// TIA Portal V18 export
FUNCTION "ChangeOverProcess" : Void   // FC1000, LAD
{ S7_Optimized_Access := 'TRUE' }
// stored: AutoNumber false, SetENOAutomatically false
   VAR_TEMP
      tBool : Bool;
   END_VAR
   VAR_TEMP   // added for the SCL form of the ladder/FBD networks
      _w1 : Bool;
      _w2 : Bool;
      _w3 : Bool;
      _w4 : Bool;
      _w5 : Bool;
      _w6 : Bool;
      _w7 : Bool;
      _w8 : Bool;
   END_VAR
BEGIN

REGION Network 1: HMI ChangeOver Confirm
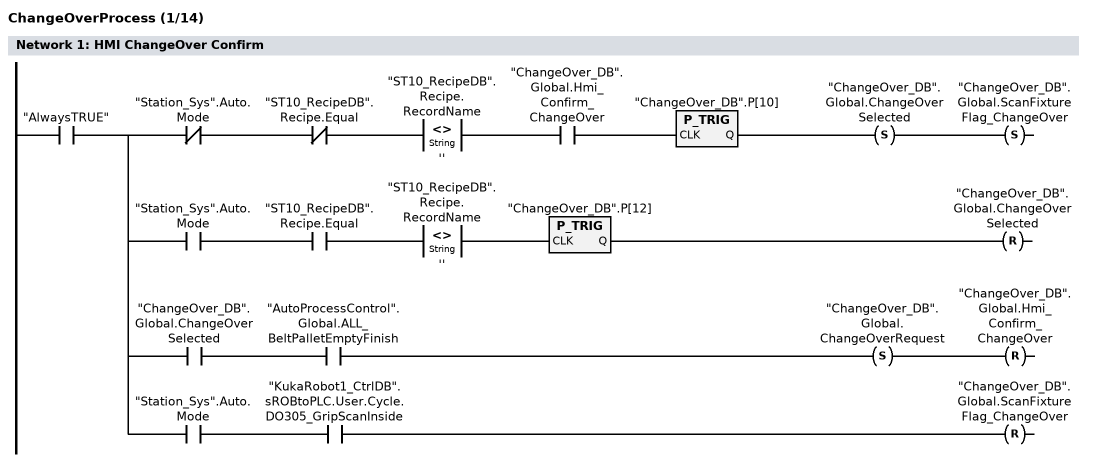
   RUNG wire#powerrail
      Contact( "AlwaysTRUE" )
      wire#w1
      I_Contact( "Station_Sys".Auto.Mode )
      I_Contact( "ST10_RecipeDB".Recipe.Equal )
      { S7_Templates := "SrcType := String" } NE_Contact(in1 := "ST10_RecipeDB".Recipe.RecordName, in2 := '')
      Contact( "ChangeOver_DB".Global.Hmi_Confirm_ChangeOver )
      P_Trig( "ChangeOver_DB".P[10] )
      S_Coil( "ChangeOver_DB".Global.ChangeOverSelected )
      S_Coil( "ChangeOver_DB".Global.ScanFixtureFlag_ChangeOver )
   END_RUNG
   RUNG wire#w1
      Contact( "Station_Sys".Auto.Mode )
      Contact( "ST10_RecipeDB".Recipe.Equal )
      { S7_Templates := "SrcType := String" } NE_Contact(in1 := "ST10_RecipeDB".Recipe.RecordName, in2 := '')
      P_Trig( "ChangeOver_DB".P[12] )
      R_Coil( "ChangeOver_DB".Global.ChangeOverSelected )
   END_RUNG
   RUNG wire#w1
      Contact( "ChangeOver_DB".Global.ChangeOverSelected )
      Contact( "AutoProcessControl".Global.ALL_BeltPalletEmptyFinish )
      S_Coil( "ChangeOver_DB".Global.ChangeOverRequest )
      R_Coil( "ChangeOver_DB".Global.Hmi_Confirm_ChangeOver )
   END_RUNG
   RUNG wire#w1
      Contact( "Station_Sys".Auto.Mode )
      Contact( "KukaRobot1_CtrlDB".sROBtoPLC.User.Cycle.DO305_GripScanInside )
      R_Coil( "ChangeOver_DB".Global.ScanFixtureFlag_ChangeOver )
   END_RUNG
   // the same network as SCL:
   #_w1 := "AlwaysTRUE" AND NOT "Station_Sys".Auto.Mode AND NOT "ST10_RecipeDB".Recipe.Equal AND ("ST10_RecipeDB".Recipe.RecordName <> '') AND "ChangeOver_DB".Global.Hmi_Confirm_ChangeOver;
   #_w2 := #_w1 AND NOT "ChangeOver_DB".P[10];   // rising edge
   "ChangeOver_DB".P[10] := #_w1;
   IF #_w2 THEN
       "ChangeOver_DB".Global.ChangeOverSelected := TRUE;
       "ChangeOver_DB".Global.ScanFixtureFlag_ChangeOver := TRUE;
   END_IF;
   #_w3 := "AlwaysTRUE" AND "Station_Sys".Auto.Mode AND "ST10_RecipeDB".Recipe.Equal AND ("ST10_RecipeDB".Recipe.RecordName <> '');
   #_w4 := #_w3 AND NOT "ChangeOver_DB".P[12];   // rising edge
   "ChangeOver_DB".P[12] := #_w3;
   IF #_w4 THEN "ChangeOver_DB".Global.ChangeOverSelected := FALSE; END_IF;
   IF "AlwaysTRUE" AND "ChangeOver_DB".Global.ChangeOverSelected AND "AutoProcessControl".Global.ALL_BeltPalletEmptyFinish THEN
       "ChangeOver_DB".Global.ChangeOverRequest := TRUE;
       "ChangeOver_DB".Global.Hmi_Confirm_ChangeOver := FALSE;
   END_IF;
   IF "AlwaysTRUE" AND "Station_Sys".Auto.Mode AND "KukaRobot1_CtrlDB".sROBtoPLC.User.Cycle.DO305_GripScanInside THEN
       "ChangeOver_DB".Global.ScanFixtureFlag_ChangeOver := FALSE;
   END_IF;
END_REGION

REGION Network 2: ChangeOverFinish Reset
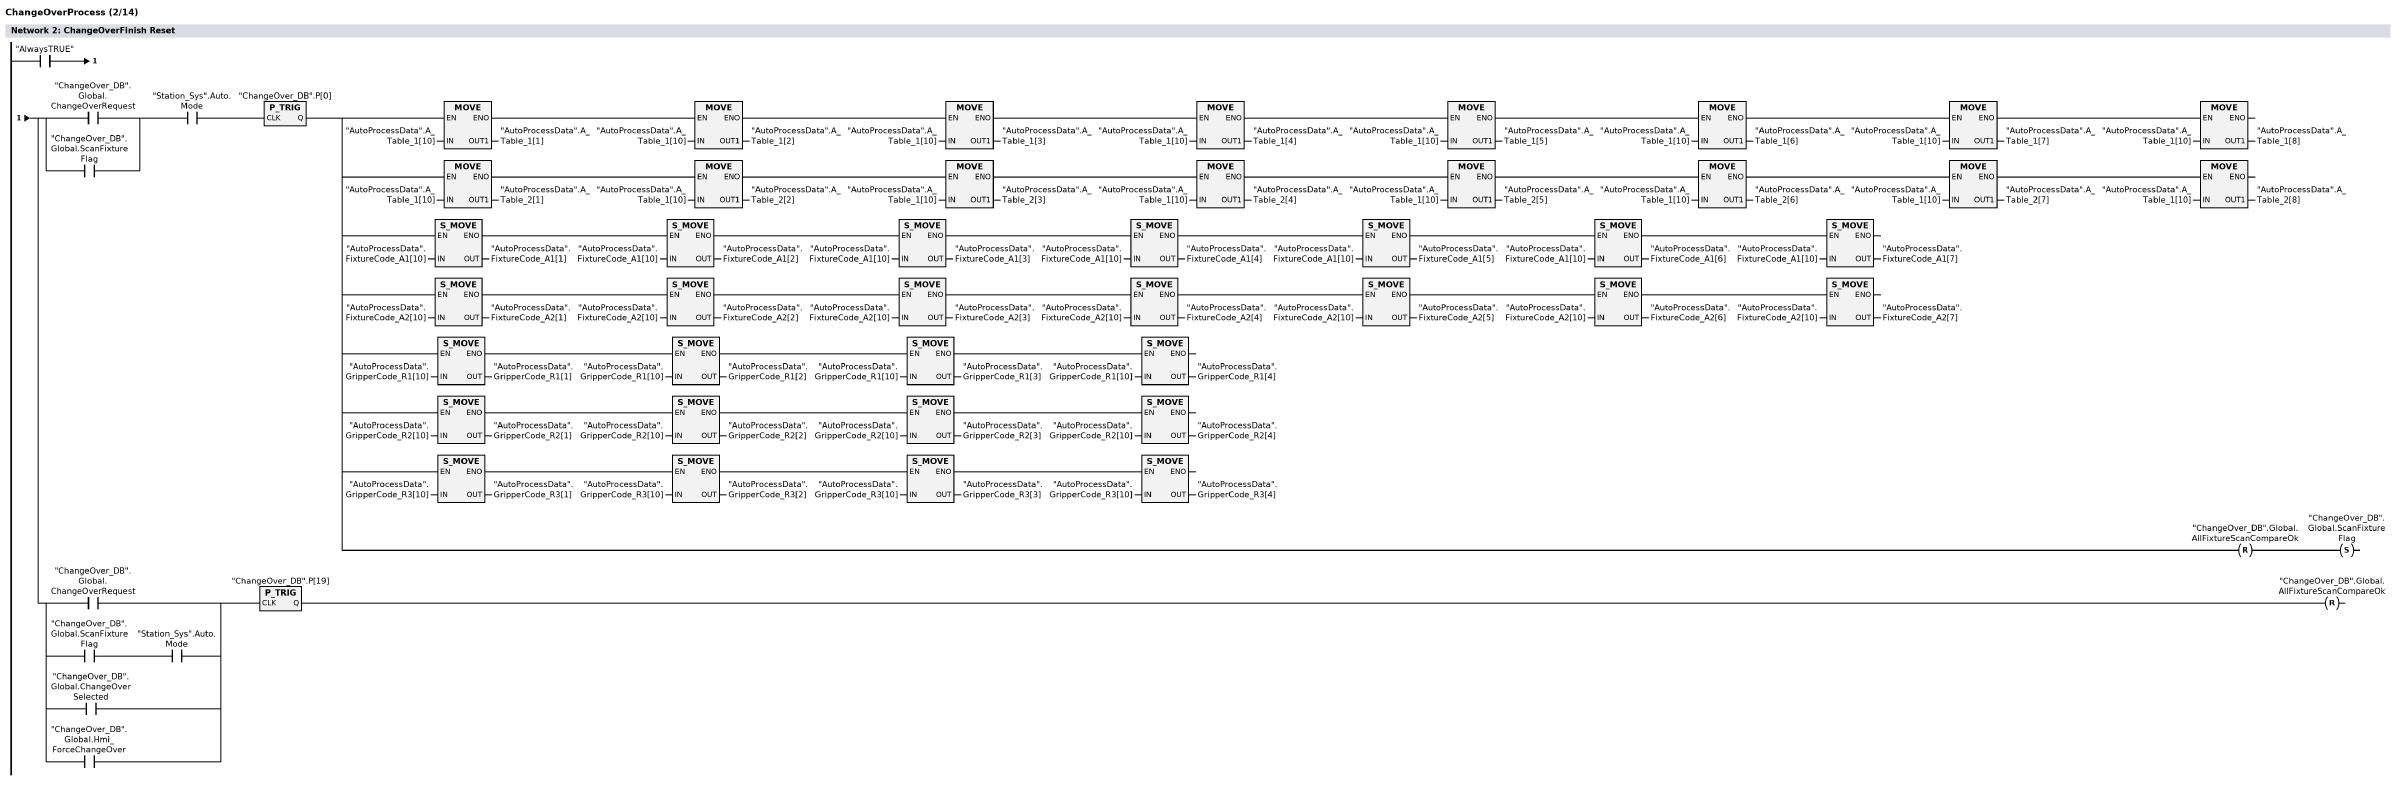
   RUNG wire#powerrail
      Contact( "AlwaysTRUE" )
      wire#w1
      Contact( "ChangeOver_DB".Global.ChangeOverRequest )
      wire#w2
      Contact( "Station_Sys".Auto.Mode )
      P_Trig( "ChangeOver_DB".P[0] )
      wire#w3
      Move(in := "AutoProcessData".A_Table_1[10], out1 => "AutoProcessData".A_Table_1[1])
      Move(in := "AutoProcessData".A_Table_1[10], out1 => "AutoProcessData".A_Table_1[2])
      Move(in := "AutoProcessData".A_Table_1[10], out1 => "AutoProcessData".A_Table_1[3])
      Move(in := "AutoProcessData".A_Table_1[10], out1 => "AutoProcessData".A_Table_1[4])
      Move(in := "AutoProcessData".A_Table_1[10], out1 => "AutoProcessData".A_Table_1[5])
      Move(in := "AutoProcessData".A_Table_1[10], out1 => "AutoProcessData".A_Table_1[6])
      Move(in := "AutoProcessData".A_Table_1[10], out1 => "AutoProcessData".A_Table_1[7])
      Move(in := "AutoProcessData".A_Table_1[10], out1 => "AutoProcessData".A_Table_1[8])
   END_RUNG
   RUNG wire#w1
      Contact( "ChangeOver_DB".Global.ScanFixtureFlag )
   END_RUNG wire#w2
   RUNG wire#w3
      Move(in := "AutoProcessData".A_Table_1[10], out1 => "AutoProcessData".A_Table_2[1])
      Move(in := "AutoProcessData".A_Table_1[10], out1 => "AutoProcessData".A_Table_2[2])
      Move(in := "AutoProcessData".A_Table_1[10], out1 => "AutoProcessData".A_Table_2[3])
      Move(in := "AutoProcessData".A_Table_1[10], out1 => "AutoProcessData".A_Table_2[4])
      Move(in := "AutoProcessData".A_Table_1[10], out1 => "AutoProcessData".A_Table_2[5])
      Move(in := "AutoProcessData".A_Table_1[10], out1 => "AutoProcessData".A_Table_2[6])
      Move(in := "AutoProcessData".A_Table_1[10], out1 => "AutoProcessData".A_Table_2[7])
      Move(in := "AutoProcessData".A_Table_1[10], out1 => "AutoProcessData".A_Table_2[8])
   END_RUNG
   RUNG wire#w3
      S_Move(in := "AutoProcessData".FixtureCode_A1[10], out => "AutoProcessData".FixtureCode_A1[1])
      S_Move(in := "AutoProcessData".FixtureCode_A1[10], out => "AutoProcessData".FixtureCode_A1[2])
      S_Move(in := "AutoProcessData".FixtureCode_A1[10], out => "AutoProcessData".FixtureCode_A1[3])
      S_Move(in := "AutoProcessData".FixtureCode_A1[10], out => "AutoProcessData".FixtureCode_A1[4])
      S_Move(in := "AutoProcessData".FixtureCode_A1[10], out => "AutoProcessData".FixtureCode_A1[5])
      S_Move(in := "AutoProcessData".FixtureCode_A1[10], out => "AutoProcessData".FixtureCode_A1[6])
      S_Move(in := "AutoProcessData".FixtureCode_A1[10], out => "AutoProcessData".FixtureCode_A1[7])
   END_RUNG
   RUNG wire#w3
      S_Move(in := "AutoProcessData".FixtureCode_A2[10], out => "AutoProcessData".FixtureCode_A2[1])
      S_Move(in := "AutoProcessData".FixtureCode_A2[10], out => "AutoProcessData".FixtureCode_A2[2])
      S_Move(in := "AutoProcessData".FixtureCode_A2[10], out => "AutoProcessData".FixtureCode_A2[3])
      S_Move(in := "AutoProcessData".FixtureCode_A2[10], out => "AutoProcessData".FixtureCode_A2[4])
      S_Move(in := "AutoProcessData".FixtureCode_A2[10], out => "AutoProcessData".FixtureCode_A2[5])
      S_Move(in := "AutoProcessData".FixtureCode_A2[10], out => "AutoProcessData".FixtureCode_A2[6])
      S_Move(in := "AutoProcessData".FixtureCode_A2[10], out => "AutoProcessData".FixtureCode_A2[7])
   END_RUNG
   RUNG wire#w3
      S_Move(in := "AutoProcessData".GripperCode_R1[10], out => "AutoProcessData".GripperCode_R1[1])
      S_Move(in := "AutoProcessData".GripperCode_R1[10], out => "AutoProcessData".GripperCode_R1[2])
      S_Move(in := "AutoProcessData".GripperCode_R1[10], out => "AutoProcessData".GripperCode_R1[3])
      S_Move(in := "AutoProcessData".GripperCode_R1[10], out => "AutoProcessData".GripperCode_R1[4])
   END_RUNG
   RUNG wire#w3
      S_Move(in := "AutoProcessData".GripperCode_R2[10], out => "AutoProcessData".GripperCode_R2[1])
      S_Move(in := "AutoProcessData".GripperCode_R2[10], out => "AutoProcessData".GripperCode_R2[2])
      S_Move(in := "AutoProcessData".GripperCode_R2[10], out => "AutoProcessData".GripperCode_R2[3])
      S_Move(in := "AutoProcessData".GripperCode_R2[10], out => "AutoProcessData".GripperCode_R2[4])
   END_RUNG
   RUNG wire#w3
      S_Move(in := "AutoProcessData".GripperCode_R3[10], out => "AutoProcessData".GripperCode_R3[1])
      S_Move(in := "AutoProcessData".GripperCode_R3[10], out => "AutoProcessData".GripperCode_R3[2])
      S_Move(in := "AutoProcessData".GripperCode_R3[10], out => "AutoProcessData".GripperCode_R3[3])
      S_Move(in := "AutoProcessData".GripperCode_R3[10], out => "AutoProcessData".GripperCode_R3[4])
   END_RUNG
   RUNG wire#w3
      R_Coil( "ChangeOver_DB".Global.AllFixtureScanCompareOk )
      S_Coil( "ChangeOver_DB".Global.ScanFixtureFlag )
   END_RUNG
   RUNG wire#w1
      Contact( "ChangeOver_DB".Global.ChangeOverRequest )
      wire#w4
      P_Trig( "ChangeOver_DB".P[19] )
      R_Coil( "ChangeOver_DB".Global.AllFixtureScanCompareOk )
   END_RUNG
   RUNG wire#w1
      Contact( "ChangeOver_DB".Global.ScanFixtureFlag )
      Contact( "Station_Sys".Auto.Mode )
   END_RUNG wire#w4
   RUNG wire#w1
      Contact( "ChangeOver_DB".Global.ChangeOverSelected )
   END_RUNG wire#w4
   RUNG wire#w1
      Contact( "ChangeOver_DB".Global.Hmi_ForceChangeOver )
   END_RUNG wire#w4
   // the same network as SCL:
   #_w1 := "AlwaysTRUE" AND ("ChangeOver_DB".Global.ChangeOverRequest OR "ChangeOver_DB".Global.ScanFixtureFlag) AND "Station_Sys".Auto.Mode;
   #_w2 := #_w1 AND NOT "ChangeOver_DB".P[0];   // rising edge
   "ChangeOver_DB".P[0] := #_w1;
   IF #_w2 THEN
       "AutoProcessData".A_Table_1[1] := "AutoProcessData".A_Table_1[10];
       "AutoProcessData".A_Table_1[2] := "AutoProcessData".A_Table_1[10];
       "AutoProcessData".A_Table_1[3] := "AutoProcessData".A_Table_1[10];
       "AutoProcessData".A_Table_1[4] := "AutoProcessData".A_Table_1[10];
       "AutoProcessData".A_Table_1[5] := "AutoProcessData".A_Table_1[10];
       "AutoProcessData".A_Table_1[6] := "AutoProcessData".A_Table_1[10];
       "AutoProcessData".A_Table_1[7] := "AutoProcessData".A_Table_1[10];
       "AutoProcessData".A_Table_1[8] := "AutoProcessData".A_Table_1[10];
       "AutoProcessData".A_Table_2[1] := "AutoProcessData".A_Table_1[10];
       "AutoProcessData".A_Table_2[2] := "AutoProcessData".A_Table_1[10];
       "AutoProcessData".A_Table_2[3] := "AutoProcessData".A_Table_1[10];
       "AutoProcessData".A_Table_2[4] := "AutoProcessData".A_Table_1[10];
       "AutoProcessData".A_Table_2[5] := "AutoProcessData".A_Table_1[10];
       "AutoProcessData".A_Table_2[6] := "AutoProcessData".A_Table_1[10];
       "AutoProcessData".A_Table_2[7] := "AutoProcessData".A_Table_1[10];
       "AutoProcessData".A_Table_2[8] := "AutoProcessData".A_Table_1[10];
       "AutoProcessData".FixtureCode_A1[1] := "AutoProcessData".FixtureCode_A1[10];
       "AutoProcessData".FixtureCode_A1[2] := "AutoProcessData".FixtureCode_A1[10];
       "AutoProcessData".FixtureCode_A1[3] := "AutoProcessData".FixtureCode_A1[10];
       "AutoProcessData".FixtureCode_A1[4] := "AutoProcessData".FixtureCode_A1[10];
       "AutoProcessData".FixtureCode_A1[5] := "AutoProcessData".FixtureCode_A1[10];
       "AutoProcessData".FixtureCode_A1[6] := "AutoProcessData".FixtureCode_A1[10];
       "AutoProcessData".FixtureCode_A1[7] := "AutoProcessData".FixtureCode_A1[10];
       "AutoProcessData".FixtureCode_A2[1] := "AutoProcessData".FixtureCode_A2[10];
       "AutoProcessData".FixtureCode_A2[2] := "AutoProcessData".FixtureCode_A2[10];
       "AutoProcessData".FixtureCode_A2[3] := "AutoProcessData".FixtureCode_A2[10];
       "AutoProcessData".FixtureCode_A2[4] := "AutoProcessData".FixtureCode_A2[10];
       "AutoProcessData".FixtureCode_A2[5] := "AutoProcessData".FixtureCode_A2[10];
       "AutoProcessData".FixtureCode_A2[6] := "AutoProcessData".FixtureCode_A2[10];
       "AutoProcessData".FixtureCode_A2[7] := "AutoProcessData".FixtureCode_A2[10];
       "AutoProcessData".GripperCode_R1[1] := "AutoProcessData".GripperCode_R1[10];
       "AutoProcessData".GripperCode_R1[2] := "AutoProcessData".GripperCode_R1[10];
       "AutoProcessData".GripperCode_R1[3] := "AutoProcessData".GripperCode_R1[10];
       "AutoProcessData".GripperCode_R1[4] := "AutoProcessData".GripperCode_R1[10];
       "AutoProcessData".GripperCode_R2[1] := "AutoProcessData".GripperCode_R2[10];
       "AutoProcessData".GripperCode_R2[2] := "AutoProcessData".GripperCode_R2[10];
       "AutoProcessData".GripperCode_R2[3] := "AutoProcessData".GripperCode_R2[10];
       "AutoProcessData".GripperCode_R2[4] := "AutoProcessData".GripperCode_R2[10];
       "AutoProcessData".GripperCode_R3[1] := "AutoProcessData".GripperCode_R3[10];
       "AutoProcessData".GripperCode_R3[2] := "AutoProcessData".GripperCode_R3[10];
       "AutoProcessData".GripperCode_R3[3] := "AutoProcessData".GripperCode_R3[10];
       "AutoProcessData".GripperCode_R3[4] := "AutoProcessData".GripperCode_R3[10];
       "ChangeOver_DB".Global.AllFixtureScanCompareOk := FALSE;
       "ChangeOver_DB".Global.ScanFixtureFlag := TRUE;
   END_IF;
   #_w3 := "AlwaysTRUE" AND ("ChangeOver_DB".Global.ChangeOverRequest OR ("ChangeOver_DB".Global.ScanFixtureFlag AND "Station_Sys".Auto.Mode) OR "ChangeOver_DB".Global.ChangeOverSelected OR "ChangeOver_DB".Global.Hmi_ForceChangeOver);
   #_w4 := #_w3 AND NOT "ChangeOver_DB".P[19];   // rising edge
   "ChangeOver_DB".P[19] := #_w3;
   IF #_w4 THEN "ChangeOver_DB".Global.AllFixtureScanCompareOk := FALSE; END_IF;
END_REGION

REGION Network 3: ManualModeFlag
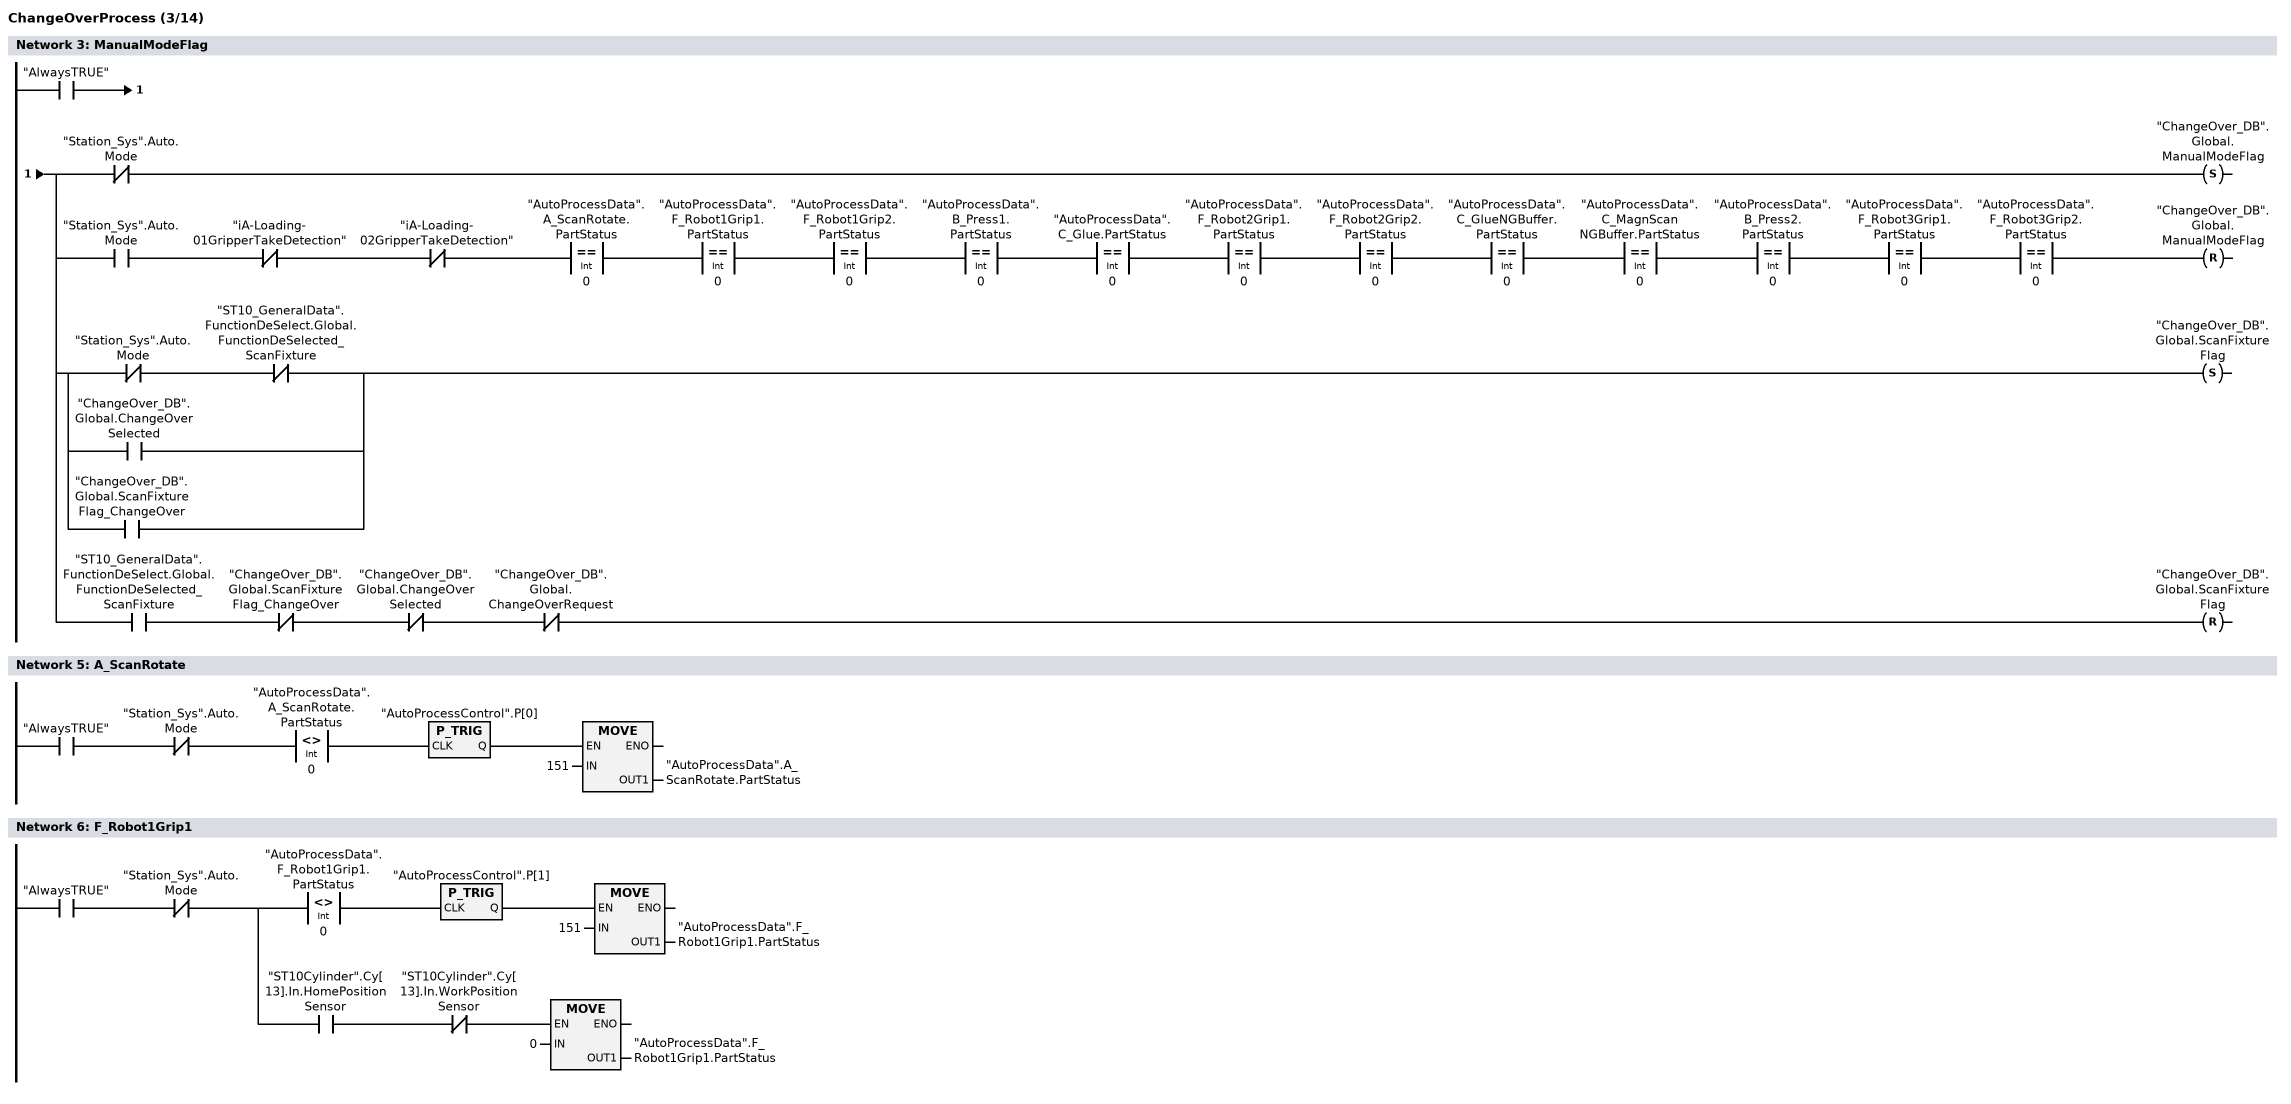
   RUNG wire#powerrail
      Contact( "AlwaysTRUE" )
      wire#w1
      I_Contact( "Station_Sys".Auto.Mode )
      S_Coil( "ChangeOver_DB".Global.ManualModeFlag )
   END_RUNG
   RUNG wire#w1
      Contact( "Station_Sys".Auto.Mode )
      I_Contact( "iA-Loading-01GripperTakeDetection" )
      I_Contact( "iA-Loading-02GripperTakeDetection" )
      { S7_Templates := "SrcType := Int" } EQ_Contact(in1 := "AutoProcessData".A_ScanRotate.PartStatus, in2 := 0)
      { S7_Templates := "SrcType := Int" } EQ_Contact(in1 := "AutoProcessData".F_Robot1Grip1.PartStatus, in2 := 0)
      { S7_Templates := "SrcType := Int" } EQ_Contact(in1 := "AutoProcessData".F_Robot1Grip2.PartStatus, in2 := 0)
      { S7_Templates := "SrcType := Int" } EQ_Contact(in1 := "AutoProcessData".B_Press1.PartStatus, in2 := 0)
      { S7_Templates := "SrcType := Int" } EQ_Contact(in1 := "AutoProcessData".C_Glue.PartStatus, in2 := 0)
      { S7_Templates := "SrcType := Int" } EQ_Contact(in1 := "AutoProcessData".F_Robot2Grip1.PartStatus, in2 := 0)
      { S7_Templates := "SrcType := Int" } EQ_Contact(in1 := "AutoProcessData".F_Robot2Grip2.PartStatus, in2 := 0)
      { S7_Templates := "SrcType := Int" } EQ_Contact(in1 := "AutoProcessData".C_GlueNGBuffer.PartStatus, in2 := 0)
      { S7_Templates := "SrcType := Int" } EQ_Contact(in1 := "AutoProcessData".C_MagnScanNGBuffer.PartStatus, in2 := 0)
      { S7_Templates := "SrcType := Int" } EQ_Contact(in1 := "AutoProcessData".B_Press2.PartStatus, in2 := 0)
      { S7_Templates := "SrcType := Int" } EQ_Contact(in1 := "AutoProcessData".F_Robot3Grip1.PartStatus, in2 := 0)
      { S7_Templates := "SrcType := Int" } EQ_Contact(in1 := "AutoProcessData".F_Robot3Grip2.PartStatus, in2 := 0)
      R_Coil( "ChangeOver_DB".Global.ManualModeFlag )
   END_RUNG
   RUNG wire#w1
      I_Contact( "Station_Sys".Auto.Mode )
      I_Contact( "ST10_GeneralData".FunctionDeSelect.Global.FunctionDeSelected_ScanFixture )
      wire#w2
      S_Coil( "ChangeOver_DB".Global.ScanFixtureFlag )
   END_RUNG
   RUNG wire#w1
      Contact( "ChangeOver_DB".Global.ChangeOverSelected )
   END_RUNG wire#w2
   RUNG wire#w1
      Contact( "ChangeOver_DB".Global.ScanFixtureFlag_ChangeOver )
   END_RUNG wire#w2
   RUNG wire#w1
      Contact( "ST10_GeneralData".FunctionDeSelect.Global.FunctionDeSelected_ScanFixture )
      I_Contact( "ChangeOver_DB".Global.ScanFixtureFlag_ChangeOver )
      I_Contact( "ChangeOver_DB".Global.ChangeOverSelected )
      I_Contact( "ChangeOver_DB".Global.ChangeOverRequest )
      R_Coil( "ChangeOver_DB".Global.ScanFixtureFlag )
   END_RUNG
   // the same network as SCL:
   IF "AlwaysTRUE" AND NOT "Station_Sys".Auto.Mode THEN
       "ChangeOver_DB".Global.ManualModeFlag := TRUE;
   END_IF;
   IF "AlwaysTRUE" AND "Station_Sys".Auto.Mode AND NOT "iA-Loading-01GripperTakeDetection" AND NOT "iA-Loading-02GripperTakeDetection" AND ("AutoProcessData".A_ScanRotate.PartStatus = 0) AND ("AutoProcessData".F_Robot1Grip1.PartStatus = 0) AND ("AutoProcessData".F_Robot1Grip2.PartStatus = 0) AND ("AutoProcessData".B_Press1.PartStatus = 0) AND ("AutoProcessData".C_Glue.PartStatus = 0) AND ("AutoProcessData".F_Robot2Grip1.PartStatus = 0) AND ("AutoProcessData".F_Robot2Grip2.PartStatus = 0) AND ("AutoProcessData".C_GlueNGBuffer.PartStatus = 0) AND ("AutoProcessData".C_MagnScanNGBuffer.PartStatus = 0) AND ("AutoProcessData".B_Press2.PartStatus = 0) AND ("AutoProcessData".F_Robot3Grip1.PartStatus = 0) AND ("AutoProcessData".F_Robot3Grip2.PartStatus = 0) THEN
       "ChangeOver_DB".Global.ManualModeFlag := FALSE;
   END_IF;
   IF "AlwaysTRUE" AND ((NOT "Station_Sys".Auto.Mode AND NOT "ST10_GeneralData".FunctionDeSelect.Global.FunctionDeSelected_ScanFixture) OR "ChangeOver_DB".Global.ChangeOverSelected OR "ChangeOver_DB".Global.ScanFixtureFlag_ChangeOver) THEN
       "ChangeOver_DB".Global.ScanFixtureFlag := TRUE;
   END_IF;
   IF "AlwaysTRUE" AND "ST10_GeneralData".FunctionDeSelect.Global.FunctionDeSelected_ScanFixture AND NOT "ChangeOver_DB".Global.ScanFixtureFlag_ChangeOver AND NOT "ChangeOver_DB".Global.ChangeOverSelected AND NOT "ChangeOver_DB".Global.ChangeOverRequest THEN
       "ChangeOver_DB".Global.ScanFixtureFlag := FALSE;
   END_IF;
END_REGION

REGION Network 4: ----------------------------- Manu Mode,All the part NG -------------------------------------------------------
END_REGION

REGION Network 5: A_ScanRotate
   RUNG wire#powerrail
      Contact( "AlwaysTRUE" )
      I_Contact( "Station_Sys".Auto.Mode )
      { S7_Templates := "SrcType := Int" } NE_Contact(in1 := "AutoProcessData".A_ScanRotate.PartStatus, in2 := 0)
      P_Trig( "AutoProcessControl".P[0] )
      Move(in := 151, out1 => "AutoProcessData".A_ScanRotate.PartStatus)
   END_RUNG
   // the same network as SCL:
   #_w1 := "AlwaysTRUE" AND NOT "Station_Sys".Auto.Mode AND ("AutoProcessData".A_ScanRotate.PartStatus <> 0);
   #_w2 := #_w1 AND NOT "AutoProcessControl".P[0];   // rising edge
   "AutoProcessControl".P[0] := #_w1;
   IF #_w2 THEN "AutoProcessData".A_ScanRotate.PartStatus := 151; END_IF;
END_REGION

REGION Network 6: F_Robot1Grip1
   RUNG wire#powerrail
      Contact( "AlwaysTRUE" )
      I_Contact( "Station_Sys".Auto.Mode )
      wire#w1
      { S7_Templates := "SrcType := Int" } NE_Contact(in1 := "AutoProcessData".F_Robot1Grip1.PartStatus, in2 := 0)
      P_Trig( "AutoProcessControl".P[1] )
      Move(in := 151, out1 => "AutoProcessData".F_Robot1Grip1.PartStatus)
   END_RUNG
   RUNG wire#w1
      Contact( "ST10Cylinder".Cy[13].In.HomePositionSensor )
      I_Contact( "ST10Cylinder".Cy[13].In.WorkPositionSensor )
      Move(in := 0, out1 => "AutoProcessData".F_Robot1Grip1.PartStatus)
   END_RUNG
   // the same network as SCL:
   #_w1 := "AlwaysTRUE" AND NOT "Station_Sys".Auto.Mode;
   #_w2 := #_w1 AND ("AutoProcessData".F_Robot1Grip1.PartStatus <> 0);
   #_w3 := #_w2 AND NOT "AutoProcessControl".P[1];   // rising edge
   "AutoProcessControl".P[1] := #_w2;
   IF #_w3 THEN "AutoProcessData".F_Robot1Grip1.PartStatus := 151; END_IF;
   IF #_w1 AND "ST10Cylinder".Cy[13].In.HomePositionSensor AND NOT "ST10Cylinder".Cy[13].In.WorkPositionSensor THEN
       "AutoProcessData".F_Robot1Grip1.PartStatus := 0;
   END_IF;
END_REGION

REGION Network 7: F_Robot1Grip2
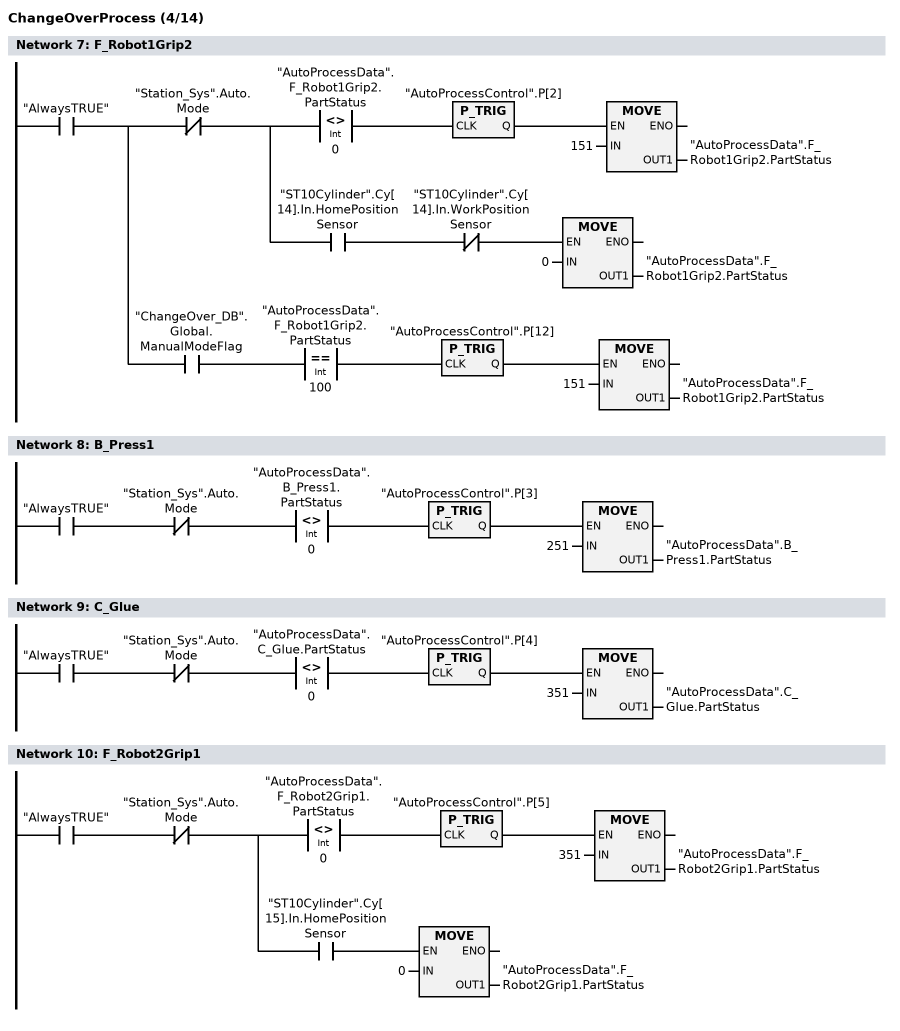
   RUNG wire#powerrail
      Contact( "AlwaysTRUE" )
      wire#w1
      I_Contact( "Station_Sys".Auto.Mode )
      wire#w2
      { S7_Templates := "SrcType := Int" } NE_Contact(in1 := "AutoProcessData".F_Robot1Grip2.PartStatus, in2 := 0)
      P_Trig( "AutoProcessControl".P[2] )
      Move(in := 151, out1 => "AutoProcessData".F_Robot1Grip2.PartStatus)
   END_RUNG
   RUNG wire#w2
      Contact( "ST10Cylinder".Cy[14].In.HomePositionSensor )
      I_Contact( "ST10Cylinder".Cy[14].In.WorkPositionSensor )
      Move(in := 0, out1 => "AutoProcessData".F_Robot1Grip2.PartStatus)
   END_RUNG
   RUNG wire#w1
      Contact( "ChangeOver_DB".Global.ManualModeFlag )
      { S7_Templates := "SrcType := Int" } EQ_Contact(in1 := "AutoProcessData".F_Robot1Grip2.PartStatus, in2 := 100)
      P_Trig( "AutoProcessControl".P[12] )
      Move(in := 151, out1 => "AutoProcessData".F_Robot1Grip2.PartStatus)
   END_RUNG
   // the same network as SCL:
   #_w1 := "AlwaysTRUE" AND NOT "Station_Sys".Auto.Mode;
   #_w2 := #_w1 AND ("AutoProcessData".F_Robot1Grip2.PartStatus <> 0);
   #_w3 := #_w2 AND NOT "AutoProcessControl".P[2];   // rising edge
   "AutoProcessControl".P[2] := #_w2;
   IF #_w3 THEN "AutoProcessData".F_Robot1Grip2.PartStatus := 151; END_IF;
   IF #_w1 AND "ST10Cylinder".Cy[14].In.HomePositionSensor AND NOT "ST10Cylinder".Cy[14].In.WorkPositionSensor THEN
       "AutoProcessData".F_Robot1Grip2.PartStatus := 0;
   END_IF;
   #_w4 := "AlwaysTRUE" AND "ChangeOver_DB".Global.ManualModeFlag AND ("AutoProcessData".F_Robot1Grip2.PartStatus = 100);
   #_w5 := #_w4 AND NOT "AutoProcessControl".P[12];   // rising edge
   "AutoProcessControl".P[12] := #_w4;
   IF #_w5 THEN "AutoProcessData".F_Robot1Grip2.PartStatus := 151; END_IF;
END_REGION

REGION Network 8: B_Press1
   RUNG wire#powerrail
      Contact( "AlwaysTRUE" )
      I_Contact( "Station_Sys".Auto.Mode )
      { S7_Templates := "SrcType := Int" } NE_Contact(in1 := "AutoProcessData".B_Press1.PartStatus, in2 := 0)
      P_Trig( "AutoProcessControl".P[3] )
      Move(in := 251, out1 => "AutoProcessData".B_Press1.PartStatus)
   END_RUNG
   // the same network as SCL:
   #_w1 := "AlwaysTRUE" AND NOT "Station_Sys".Auto.Mode AND ("AutoProcessData".B_Press1.PartStatus <> 0);
   #_w2 := #_w1 AND NOT "AutoProcessControl".P[3];   // rising edge
   "AutoProcessControl".P[3] := #_w1;
   IF #_w2 THEN "AutoProcessData".B_Press1.PartStatus := 251; END_IF;
END_REGION

REGION Network 9: C_Glue
   RUNG wire#powerrail
      Contact( "AlwaysTRUE" )
      I_Contact( "Station_Sys".Auto.Mode )
      { S7_Templates := "SrcType := Int" } NE_Contact(in1 := "AutoProcessData".C_Glue.PartStatus, in2 := 0)
      P_Trig( "AutoProcessControl".P[4] )
      Move(in := 351, out1 => "AutoProcessData".C_Glue.PartStatus)
   END_RUNG
   // the same network as SCL:
   #_w1 := "AlwaysTRUE" AND NOT "Station_Sys".Auto.Mode AND ("AutoProcessData".C_Glue.PartStatus <> 0);
   #_w2 := #_w1 AND NOT "AutoProcessControl".P[4];   // rising edge
   "AutoProcessControl".P[4] := #_w1;
   IF #_w2 THEN "AutoProcessData".C_Glue.PartStatus := 351; END_IF;
END_REGION

REGION Network 10: F_Robot2Grip1
   RUNG wire#powerrail
      Contact( "AlwaysTRUE" )
      I_Contact( "Station_Sys".Auto.Mode )
      wire#w1
      { S7_Templates := "SrcType := Int" } NE_Contact(in1 := "AutoProcessData".F_Robot2Grip1.PartStatus, in2 := 0)
      P_Trig( "AutoProcessControl".P[5] )
      Move(in := 351, out1 => "AutoProcessData".F_Robot2Grip1.PartStatus)
   END_RUNG
   RUNG wire#w1
      Contact( "ST10Cylinder".Cy[15].In.HomePositionSensor )
      Move(in := 0, out1 => "AutoProcessData".F_Robot2Grip1.PartStatus)
   END_RUNG
   // the same network as SCL:
   #_w1 := "AlwaysTRUE" AND NOT "Station_Sys".Auto.Mode;
   #_w2 := #_w1 AND ("AutoProcessData".F_Robot2Grip1.PartStatus <> 0);
   #_w3 := #_w2 AND NOT "AutoProcessControl".P[5];   // rising edge
   "AutoProcessControl".P[5] := #_w2;
   IF #_w3 THEN "AutoProcessData".F_Robot2Grip1.PartStatus := 351; END_IF;
   IF #_w1 AND "ST10Cylinder".Cy[15].In.HomePositionSensor THEN
       "AutoProcessData".F_Robot2Grip1.PartStatus := 0;
   END_IF;
END_REGION

REGION Network 11: F_Robot2Grip2
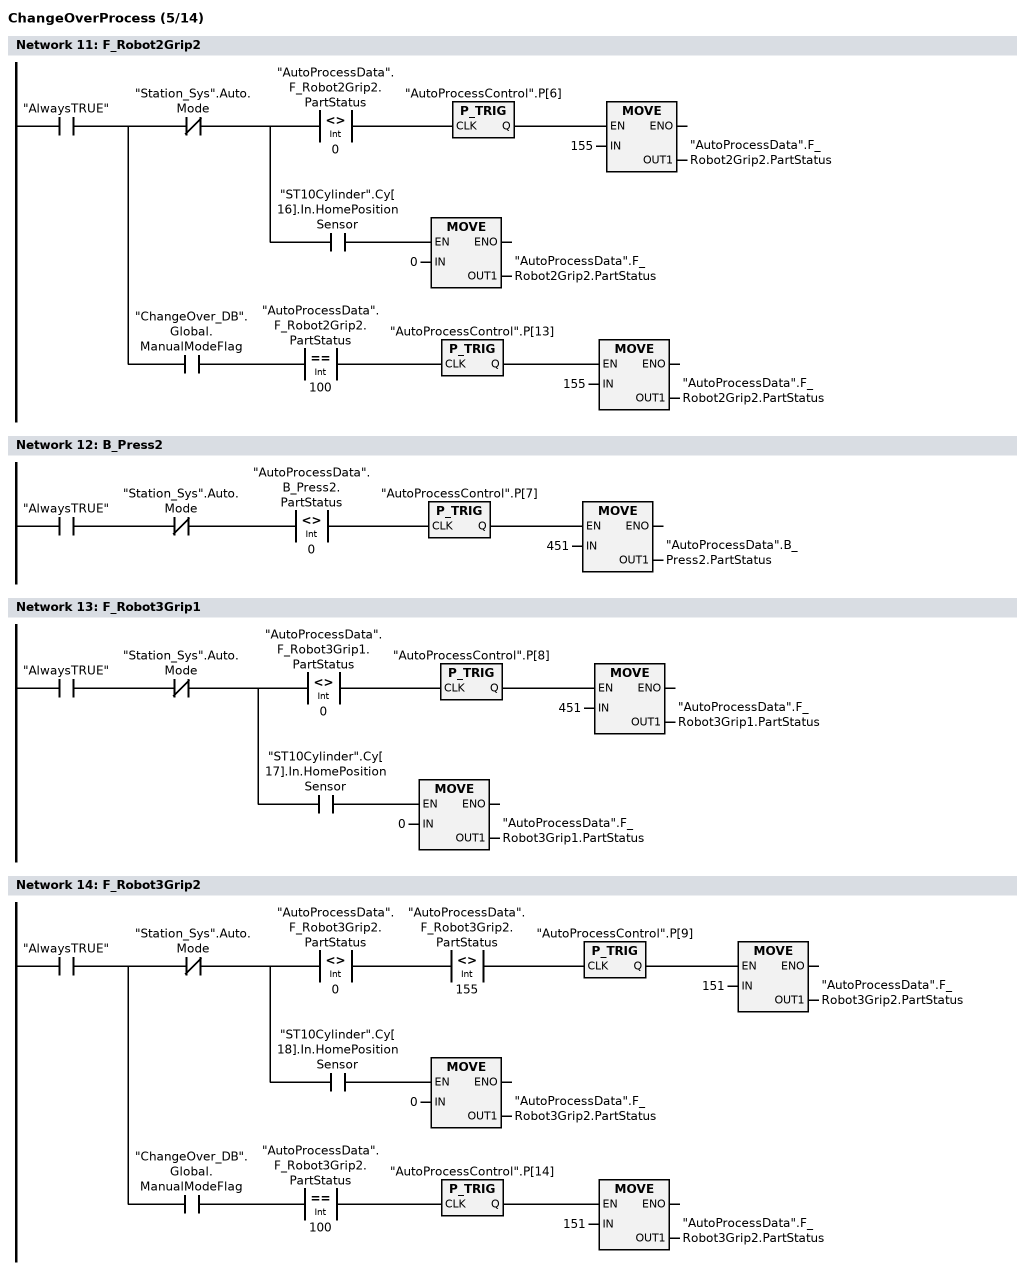
   RUNG wire#powerrail
      Contact( "AlwaysTRUE" )
      wire#w1
      I_Contact( "Station_Sys".Auto.Mode )
      wire#w2
      { S7_Templates := "SrcType := Int" } NE_Contact(in1 := "AutoProcessData".F_Robot2Grip2.PartStatus, in2 := 0)
      P_Trig( "AutoProcessControl".P[6] )
      Move(in := 155, out1 => "AutoProcessData".F_Robot2Grip2.PartStatus)
   END_RUNG
   RUNG wire#w2
      Contact( "ST10Cylinder".Cy[16].In.HomePositionSensor )
      Move(in := 0, out1 => "AutoProcessData".F_Robot2Grip2.PartStatus)
   END_RUNG
   RUNG wire#w1
      Contact( "ChangeOver_DB".Global.ManualModeFlag )
      { S7_Templates := "SrcType := Int" } EQ_Contact(in1 := "AutoProcessData".F_Robot2Grip2.PartStatus, in2 := 100)
      P_Trig( "AutoProcessControl".P[13] )
      Move(in := 155, out1 => "AutoProcessData".F_Robot2Grip2.PartStatus)
   END_RUNG
   // the same network as SCL:
   #_w1 := "AlwaysTRUE" AND NOT "Station_Sys".Auto.Mode;
   #_w2 := #_w1 AND ("AutoProcessData".F_Robot2Grip2.PartStatus <> 0);
   #_w3 := #_w2 AND NOT "AutoProcessControl".P[6];   // rising edge
   "AutoProcessControl".P[6] := #_w2;
   IF #_w3 THEN "AutoProcessData".F_Robot2Grip2.PartStatus := 155; END_IF;
   IF #_w1 AND "ST10Cylinder".Cy[16].In.HomePositionSensor THEN
       "AutoProcessData".F_Robot2Grip2.PartStatus := 0;
   END_IF;
   #_w4 := "AlwaysTRUE" AND "ChangeOver_DB".Global.ManualModeFlag AND ("AutoProcessData".F_Robot2Grip2.PartStatus = 100);
   #_w5 := #_w4 AND NOT "AutoProcessControl".P[13];   // rising edge
   "AutoProcessControl".P[13] := #_w4;
   IF #_w5 THEN "AutoProcessData".F_Robot2Grip2.PartStatus := 155; END_IF;
END_REGION

REGION Network 12: B_Press2
   RUNG wire#powerrail
      Contact( "AlwaysTRUE" )
      I_Contact( "Station_Sys".Auto.Mode )
      { S7_Templates := "SrcType := Int" } NE_Contact(in1 := "AutoProcessData".B_Press2.PartStatus, in2 := 0)
      P_Trig( "AutoProcessControl".P[7] )
      Move(in := 451, out1 => "AutoProcessData".B_Press2.PartStatus)
   END_RUNG
   // the same network as SCL:
   #_w1 := "AlwaysTRUE" AND NOT "Station_Sys".Auto.Mode AND ("AutoProcessData".B_Press2.PartStatus <> 0);
   #_w2 := #_w1 AND NOT "AutoProcessControl".P[7];   // rising edge
   "AutoProcessControl".P[7] := #_w1;
   IF #_w2 THEN "AutoProcessData".B_Press2.PartStatus := 451; END_IF;
END_REGION

REGION Network 13: F_Robot3Grip1
   RUNG wire#powerrail
      Contact( "AlwaysTRUE" )
      I_Contact( "Station_Sys".Auto.Mode )
      wire#w1
      { S7_Templates := "SrcType := Int" } NE_Contact(in1 := "AutoProcessData".F_Robot3Grip1.PartStatus, in2 := 0)
      P_Trig( "AutoProcessControl".P[8] )
      Move(in := 451, out1 => "AutoProcessData".F_Robot3Grip1.PartStatus)
   END_RUNG
   RUNG wire#w1
      Contact( "ST10Cylinder".Cy[17].In.HomePositionSensor )
      Move(in := 0, out1 => "AutoProcessData".F_Robot3Grip1.PartStatus)
   END_RUNG
   // the same network as SCL:
   #_w1 := "AlwaysTRUE" AND NOT "Station_Sys".Auto.Mode;
   #_w2 := #_w1 AND ("AutoProcessData".F_Robot3Grip1.PartStatus <> 0);
   #_w3 := #_w2 AND NOT "AutoProcessControl".P[8];   // rising edge
   "AutoProcessControl".P[8] := #_w2;
   IF #_w3 THEN "AutoProcessData".F_Robot3Grip1.PartStatus := 451; END_IF;
   IF #_w1 AND "ST10Cylinder".Cy[17].In.HomePositionSensor THEN
       "AutoProcessData".F_Robot3Grip1.PartStatus := 0;
   END_IF;
END_REGION

REGION Network 14: F_Robot3Grip2
   RUNG wire#powerrail
      Contact( "AlwaysTRUE" )
      wire#w1
      I_Contact( "Station_Sys".Auto.Mode )
      wire#w2
      { S7_Templates := "SrcType := Int" } NE_Contact(in1 := "AutoProcessData".F_Robot3Grip2.PartStatus, in2 := 0)
      { S7_Templates := "SrcType := Int" } NE_Contact(in1 := "AutoProcessData".F_Robot3Grip2.PartStatus, in2 := 155)
      P_Trig( "AutoProcessControl".P[9] )
      Move(in := 151, out1 => "AutoProcessData".F_Robot3Grip2.PartStatus)
   END_RUNG
   RUNG wire#w2
      Contact( "ST10Cylinder".Cy[18].In.HomePositionSensor )
      Move(in := 0, out1 => "AutoProcessData".F_Robot3Grip2.PartStatus)
   END_RUNG
   RUNG wire#w1
      Contact( "ChangeOver_DB".Global.ManualModeFlag )
      { S7_Templates := "SrcType := Int" } EQ_Contact(in1 := "AutoProcessData".F_Robot3Grip2.PartStatus, in2 := 100)
      P_Trig( "AutoProcessControl".P[14] )
      Move(in := 151, out1 => "AutoProcessData".F_Robot3Grip2.PartStatus)
   END_RUNG
   // the same network as SCL:
   #_w1 := "AlwaysTRUE" AND NOT "Station_Sys".Auto.Mode;
   #_w2 := #_w1 AND ("AutoProcessData".F_Robot3Grip2.PartStatus <> 0) AND ("AutoProcessData".F_Robot3Grip2.PartStatus <> 155);
   #_w3 := #_w2 AND NOT "AutoProcessControl".P[9];   // rising edge
   "AutoProcessControl".P[9] := #_w2;
   IF #_w3 THEN "AutoProcessData".F_Robot3Grip2.PartStatus := 151; END_IF;
   IF #_w1 AND "ST10Cylinder".Cy[18].In.HomePositionSensor THEN
       "AutoProcessData".F_Robot3Grip2.PartStatus := 0;
   END_IF;
   #_w4 := "AlwaysTRUE" AND "ChangeOver_DB".Global.ManualModeFlag AND ("AutoProcessData".F_Robot3Grip2.PartStatus = 100);
   #_w5 := #_w4 AND NOT "AutoProcessControl".P[14];   // rising edge
   "AutoProcessControl".P[14] := #_w4;
   IF #_w5 THEN "AutoProcessData".F_Robot3Grip2.PartStatus := 151; END_IF;
END_REGION

REGION Network 15: ---------------------------------- FixtureCode ------------------------------------------
END_REGION

REGION Network 16: A1_Table
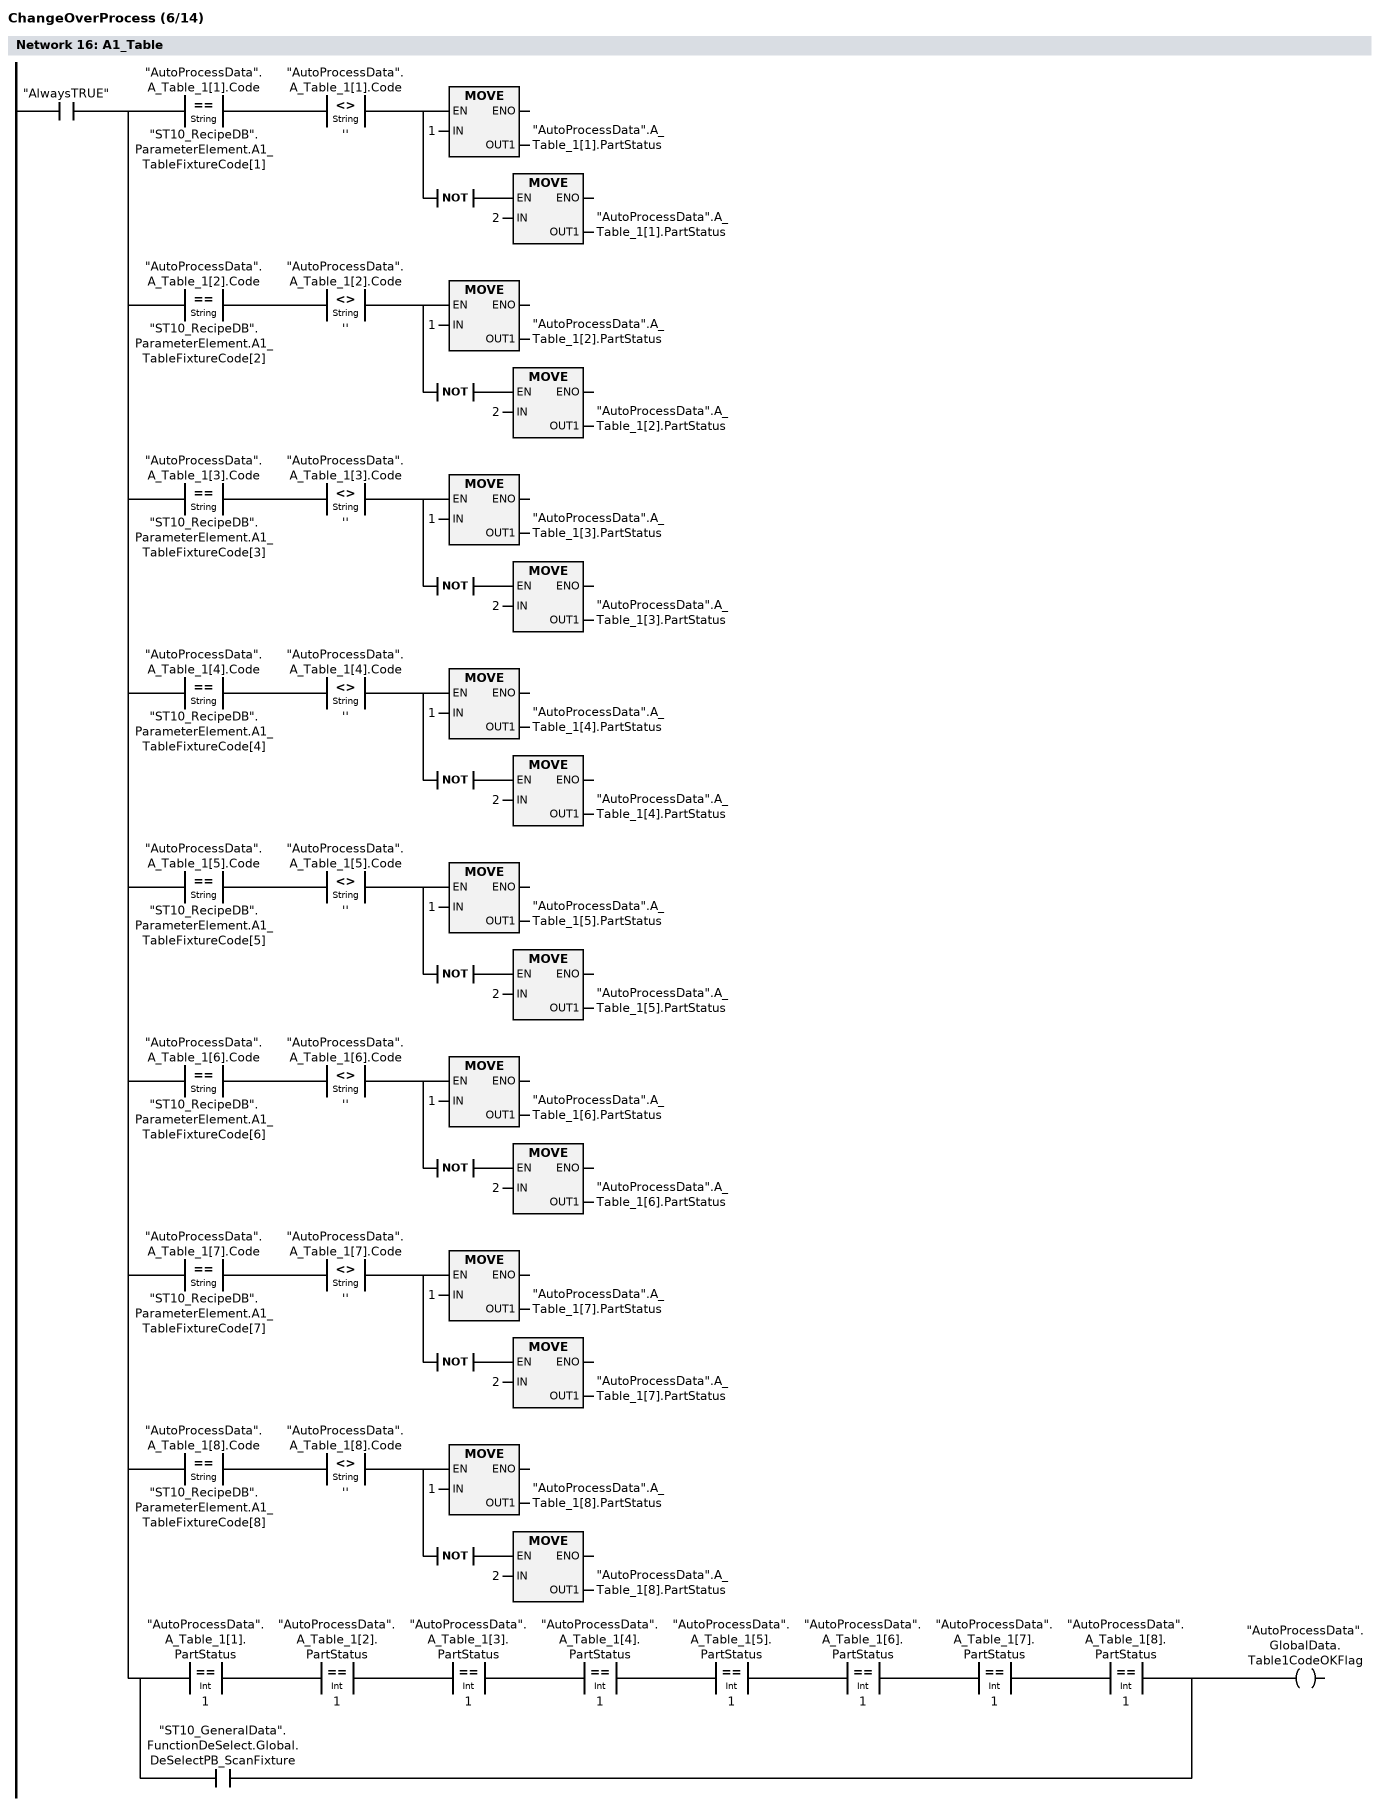
   RUNG wire#powerrail
      Contact( "AlwaysTRUE" )
      wire#w1
      { S7_Templates := "SrcType := String" } EQ_Contact(in1 := "AutoProcessData".A_Table_1[1].Code, in2 := "ST10_RecipeDB".ParameterElement.A1_TableFixtureCode[1])
      { S7_Templates := "SrcType := String" } NE_Contact(in1 := "AutoProcessData".A_Table_1[1].Code, in2 := '')
      wire#w2
      Move(in := 1, out1 => "AutoProcessData".A_Table_1[1].PartStatus)
   END_RUNG
   RUNG wire#w2
      Not()
      Move(in := 2, out1 => "AutoProcessData".A_Table_1[1].PartStatus)
   END_RUNG
   RUNG wire#w1
      { S7_Templates := "SrcType := String" } EQ_Contact(in1 := "AutoProcessData".A_Table_1[2].Code, in2 := "ST10_RecipeDB".ParameterElement.A1_TableFixtureCode[2])
      { S7_Templates := "SrcType := String" } NE_Contact(in1 := "AutoProcessData".A_Table_1[2].Code, in2 := '')
      wire#w3
      Move(in := 1, out1 => "AutoProcessData".A_Table_1[2].PartStatus)
   END_RUNG
   RUNG wire#w3
      Not()
      Move(in := 2, out1 => "AutoProcessData".A_Table_1[2].PartStatus)
   END_RUNG
   RUNG wire#w1
      { S7_Templates := "SrcType := String" } EQ_Contact(in1 := "AutoProcessData".A_Table_1[3].Code, in2 := "ST10_RecipeDB".ParameterElement.A1_TableFixtureCode[3])
      { S7_Templates := "SrcType := String" } NE_Contact(in1 := "AutoProcessData".A_Table_1[3].Code, in2 := '')
      wire#w4
      Move(in := 1, out1 => "AutoProcessData".A_Table_1[3].PartStatus)
   END_RUNG
   RUNG wire#w4
      Not()
      Move(in := 2, out1 => "AutoProcessData".A_Table_1[3].PartStatus)
   END_RUNG
   RUNG wire#w1
      { S7_Templates := "SrcType := String" } EQ_Contact(in1 := "AutoProcessData".A_Table_1[4].Code, in2 := "ST10_RecipeDB".ParameterElement.A1_TableFixtureCode[4])
      { S7_Templates := "SrcType := String" } NE_Contact(in1 := "AutoProcessData".A_Table_1[4].Code, in2 := '')
      wire#w5
      Move(in := 1, out1 => "AutoProcessData".A_Table_1[4].PartStatus)
   END_RUNG
   RUNG wire#w5
      Not()
      Move(in := 2, out1 => "AutoProcessData".A_Table_1[4].PartStatus)
   END_RUNG
   RUNG wire#w1
      { S7_Templates := "SrcType := String" } EQ_Contact(in1 := "AutoProcessData".A_Table_1[5].Code, in2 := "ST10_RecipeDB".ParameterElement.A1_TableFixtureCode[5])
      { S7_Templates := "SrcType := String" } NE_Contact(in1 := "AutoProcessData".A_Table_1[5].Code, in2 := '')
      wire#w6
      Move(in := 1, out1 => "AutoProcessData".A_Table_1[5].PartStatus)
   END_RUNG
   RUNG wire#w6
      Not()
      Move(in := 2, out1 => "AutoProcessData".A_Table_1[5].PartStatus)
   END_RUNG
   RUNG wire#w1
      { S7_Templates := "SrcType := String" } EQ_Contact(in1 := "AutoProcessData".A_Table_1[6].Code, in2 := "ST10_RecipeDB".ParameterElement.A1_TableFixtureCode[6])
      { S7_Templates := "SrcType := String" } NE_Contact(in1 := "AutoProcessData".A_Table_1[6].Code, in2 := '')
      wire#w7
      Move(in := 1, out1 => "AutoProcessData".A_Table_1[6].PartStatus)
   END_RUNG
   RUNG wire#w7
      Not()
      Move(in := 2, out1 => "AutoProcessData".A_Table_1[6].PartStatus)
   END_RUNG
   RUNG wire#w1
      { S7_Templates := "SrcType := String" } EQ_Contact(in1 := "AutoProcessData".A_Table_1[7].Code, in2 := "ST10_RecipeDB".ParameterElement.A1_TableFixtureCode[7])
      { S7_Templates := "SrcType := String" } NE_Contact(in1 := "AutoProcessData".A_Table_1[7].Code, in2 := '')
      wire#w8
      Move(in := 1, out1 => "AutoProcessData".A_Table_1[7].PartStatus)
   END_RUNG
   RUNG wire#w8
      Not()
      Move(in := 2, out1 => "AutoProcessData".A_Table_1[7].PartStatus)
   END_RUNG
   RUNG wire#w1
      { S7_Templates := "SrcType := String" } EQ_Contact(in1 := "AutoProcessData".A_Table_1[8].Code, in2 := "ST10_RecipeDB".ParameterElement.A1_TableFixtureCode[8])
      { S7_Templates := "SrcType := String" } NE_Contact(in1 := "AutoProcessData".A_Table_1[8].Code, in2 := '')
      wire#w9
      Move(in := 1, out1 => "AutoProcessData".A_Table_1[8].PartStatus)
   END_RUNG
   RUNG wire#w9
      Not()
      Move(in := 2, out1 => "AutoProcessData".A_Table_1[8].PartStatus)
   END_RUNG
   RUNG wire#w1
      { S7_Templates := "SrcType := Int" } EQ_Contact(in1 := "AutoProcessData".A_Table_1[1].PartStatus, in2 := 1)
      { S7_Templates := "SrcType := Int" } EQ_Contact(in1 := "AutoProcessData".A_Table_1[2].PartStatus, in2 := 1)
      { S7_Templates := "SrcType := Int" } EQ_Contact(in1 := "AutoProcessData".A_Table_1[3].PartStatus, in2 := 1)
      { S7_Templates := "SrcType := Int" } EQ_Contact(in1 := "AutoProcessData".A_Table_1[4].PartStatus, in2 := 1)
      { S7_Templates := "SrcType := Int" } EQ_Contact(in1 := "AutoProcessData".A_Table_1[5].PartStatus, in2 := 1)
      { S7_Templates := "SrcType := Int" } EQ_Contact(in1 := "AutoProcessData".A_Table_1[6].PartStatus, in2 := 1)
      { S7_Templates := "SrcType := Int" } EQ_Contact(in1 := "AutoProcessData".A_Table_1[7].PartStatus, in2 := 1)
      { S7_Templates := "SrcType := Int" } EQ_Contact(in1 := "AutoProcessData".A_Table_1[8].PartStatus, in2 := 1)
      wire#w10
      Coil( "AutoProcessData".GlobalData.Table1CodeOKFlag )
   END_RUNG
   RUNG wire#w1
      Contact( "ST10_GeneralData".FunctionDeSelect.Global.DeSelectPB_ScanFixture )
   END_RUNG wire#w10
   // the same network as SCL:
   #_w1 := "AlwaysTRUE" AND ("AutoProcessData".A_Table_1[1].Code = "ST10_RecipeDB".ParameterElement.A1_TableFixtureCode[1]) AND ("AutoProcessData".A_Table_1[1].Code <> '');
   IF #_w1 THEN "AutoProcessData".A_Table_1[1].PartStatus := 1; END_IF;
   IF NOT #_w1 THEN "AutoProcessData".A_Table_1[1].PartStatus := 2; END_IF;
   #_w2 := "AlwaysTRUE" AND ("AutoProcessData".A_Table_1[2].Code = "ST10_RecipeDB".ParameterElement.A1_TableFixtureCode[2]) AND ("AutoProcessData".A_Table_1[2].Code <> '');
   IF #_w2 THEN "AutoProcessData".A_Table_1[2].PartStatus := 1; END_IF;
   IF NOT #_w2 THEN "AutoProcessData".A_Table_1[2].PartStatus := 2; END_IF;
   #_w3 := "AlwaysTRUE" AND ("AutoProcessData".A_Table_1[3].Code = "ST10_RecipeDB".ParameterElement.A1_TableFixtureCode[3]) AND ("AutoProcessData".A_Table_1[3].Code <> '');
   IF #_w3 THEN "AutoProcessData".A_Table_1[3].PartStatus := 1; END_IF;
   IF NOT #_w3 THEN "AutoProcessData".A_Table_1[3].PartStatus := 2; END_IF;
   #_w4 := "AlwaysTRUE" AND ("AutoProcessData".A_Table_1[4].Code = "ST10_RecipeDB".ParameterElement.A1_TableFixtureCode[4]) AND ("AutoProcessData".A_Table_1[4].Code <> '');
   IF #_w4 THEN "AutoProcessData".A_Table_1[4].PartStatus := 1; END_IF;
   IF NOT #_w4 THEN "AutoProcessData".A_Table_1[4].PartStatus := 2; END_IF;
   #_w5 := "AlwaysTRUE" AND ("AutoProcessData".A_Table_1[5].Code = "ST10_RecipeDB".ParameterElement.A1_TableFixtureCode[5]) AND ("AutoProcessData".A_Table_1[5].Code <> '');
   IF #_w5 THEN "AutoProcessData".A_Table_1[5].PartStatus := 1; END_IF;
   IF NOT #_w5 THEN "AutoProcessData".A_Table_1[5].PartStatus := 2; END_IF;
   #_w6 := "AlwaysTRUE" AND ("AutoProcessData".A_Table_1[6].Code = "ST10_RecipeDB".ParameterElement.A1_TableFixtureCode[6]) AND ("AutoProcessData".A_Table_1[6].Code <> '');
   IF #_w6 THEN "AutoProcessData".A_Table_1[6].PartStatus := 1; END_IF;
   IF NOT #_w6 THEN "AutoProcessData".A_Table_1[6].PartStatus := 2; END_IF;
   #_w7 := "AlwaysTRUE" AND ("AutoProcessData".A_Table_1[7].Code = "ST10_RecipeDB".ParameterElement.A1_TableFixtureCode[7]) AND ("AutoProcessData".A_Table_1[7].Code <> '');
   IF #_w7 THEN "AutoProcessData".A_Table_1[7].PartStatus := 1; END_IF;
   IF NOT #_w7 THEN "AutoProcessData".A_Table_1[7].PartStatus := 2; END_IF;
   #_w8 := "AlwaysTRUE" AND ("AutoProcessData".A_Table_1[8].Code = "ST10_RecipeDB".ParameterElement.A1_TableFixtureCode[8]) AND ("AutoProcessData".A_Table_1[8].Code <> '');
   IF #_w8 THEN "AutoProcessData".A_Table_1[8].PartStatus := 1; END_IF;
   IF NOT #_w8 THEN "AutoProcessData".A_Table_1[8].PartStatus := 2; END_IF;
   "AutoProcessData".GlobalData.Table1CodeOKFlag := "AlwaysTRUE" AND ((("AutoProcessData".A_Table_1[1].PartStatus = 1) AND ("AutoProcessData".A_Table_1[2].PartStatus = 1) AND ("AutoProcessData".A_Table_1[3].PartStatus = 1) AND ("AutoProcessData".A_Table_1[4].PartStatus = 1) AND ("AutoProcessData".A_Table_1[5].PartStatus = 1) AND ("AutoProcessData".A_Table_1[6].PartStatus = 1) AND ("AutoProcessData".A_Table_1[7].PartStatus = 1) AND ("AutoProcessData".A_Table_1[8].PartStatus = 1)) OR "ST10_GeneralData".FunctionDeSelect.Global.DeSelectPB_ScanFixture);
END_REGION

REGION Network 17: A2_Table
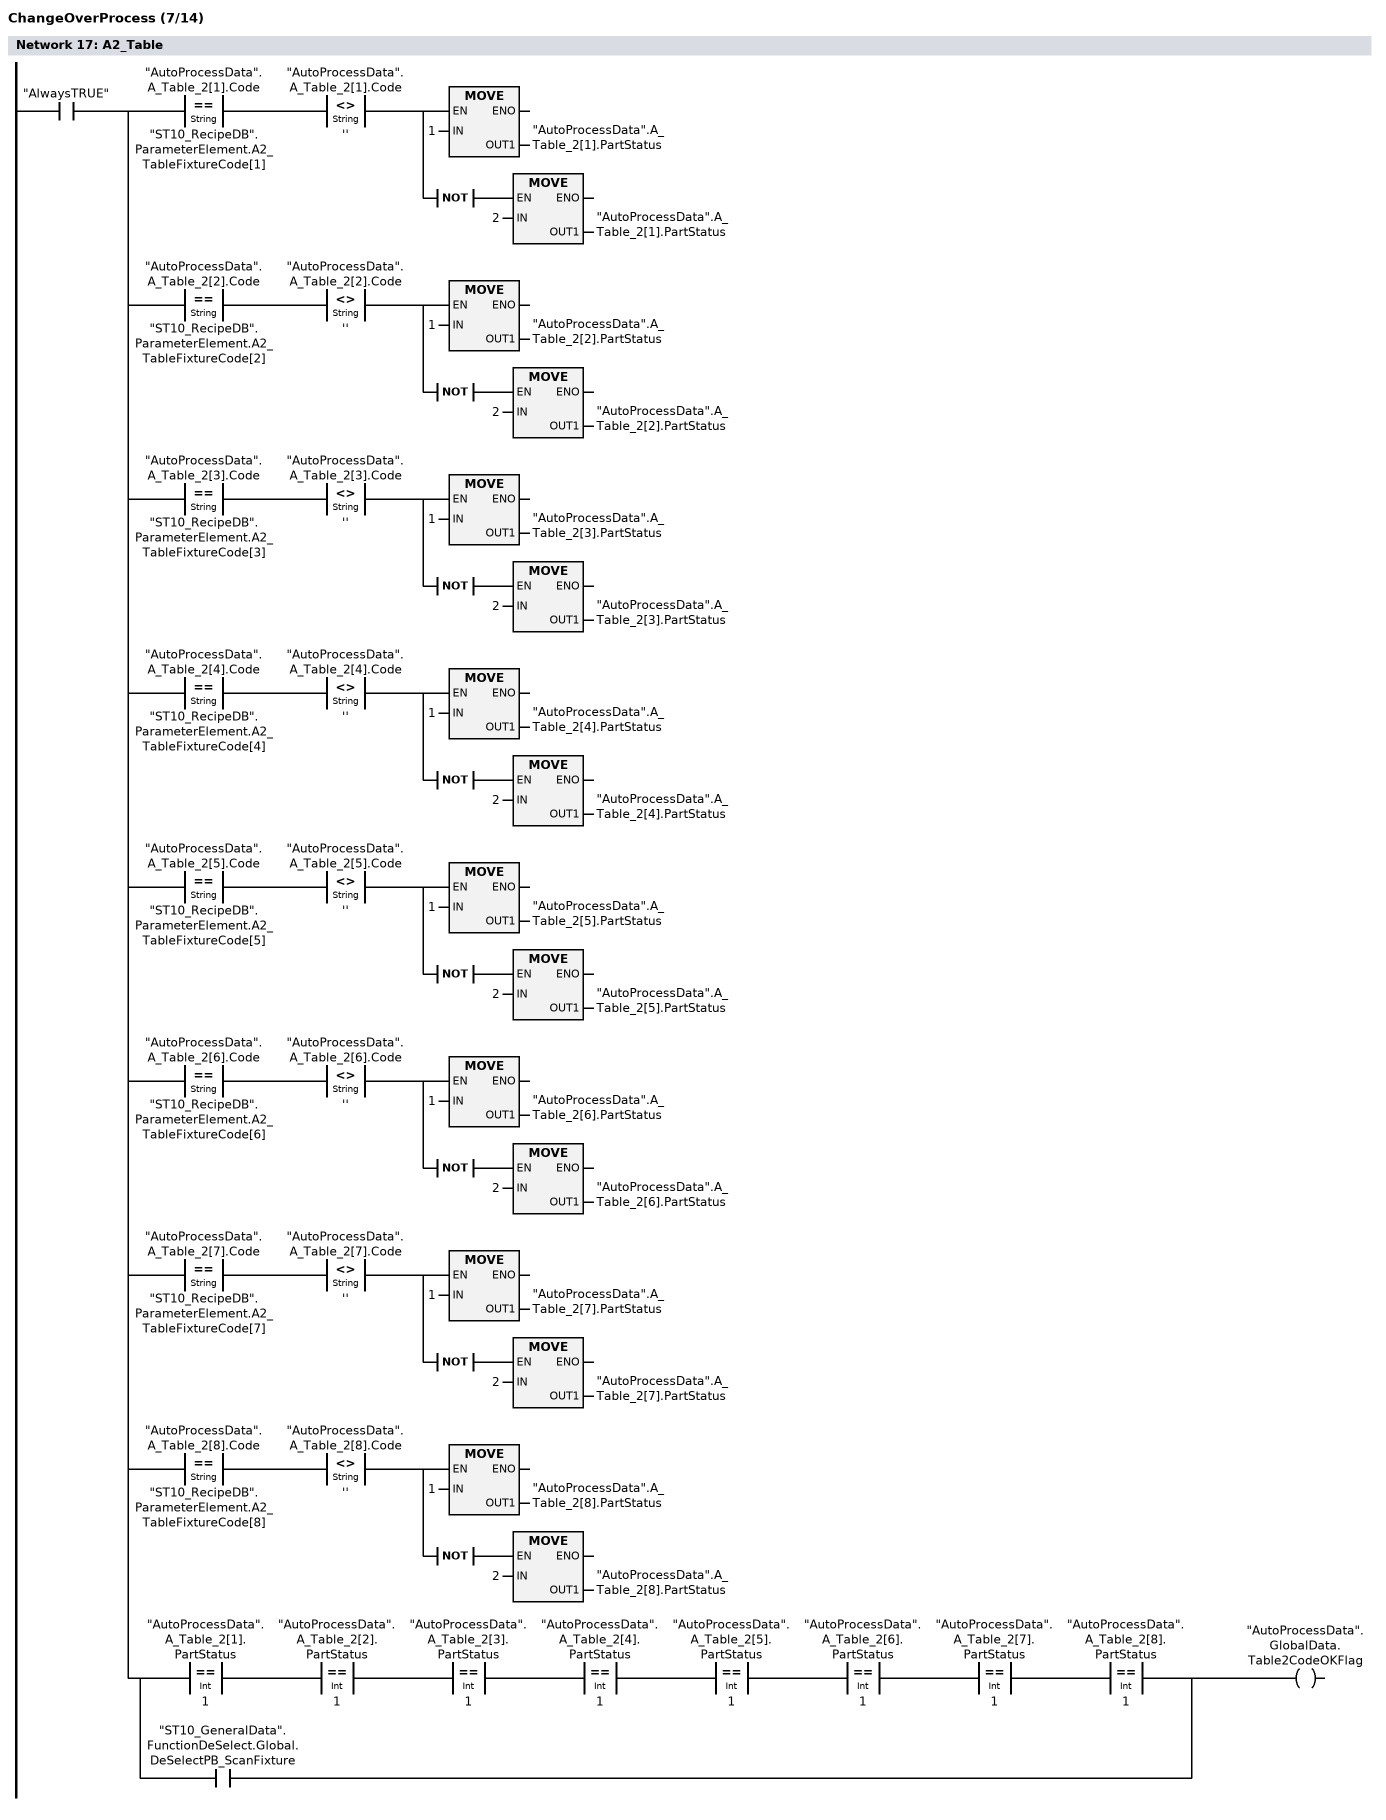
   RUNG wire#powerrail
      Contact( "AlwaysTRUE" )
      wire#w1
      { S7_Templates := "SrcType := String" } EQ_Contact(in1 := "AutoProcessData".A_Table_2[1].Code, in2 := "ST10_RecipeDB".ParameterElement.A2_TableFixtureCode[1])
      { S7_Templates := "SrcType := String" } NE_Contact(in1 := "AutoProcessData".A_Table_2[1].Code, in2 := '')
      wire#w2
      Move(in := 1, out1 => "AutoProcessData".A_Table_2[1].PartStatus)
   END_RUNG
   RUNG wire#w2
      Not()
      Move(in := 2, out1 => "AutoProcessData".A_Table_2[1].PartStatus)
   END_RUNG
   RUNG wire#w1
      { S7_Templates := "SrcType := String" } EQ_Contact(in1 := "AutoProcessData".A_Table_2[2].Code, in2 := "ST10_RecipeDB".ParameterElement.A2_TableFixtureCode[2])
      { S7_Templates := "SrcType := String" } NE_Contact(in1 := "AutoProcessData".A_Table_2[2].Code, in2 := '')
      wire#w3
      Move(in := 1, out1 => "AutoProcessData".A_Table_2[2].PartStatus)
   END_RUNG
   RUNG wire#w3
      Not()
      Move(in := 2, out1 => "AutoProcessData".A_Table_2[2].PartStatus)
   END_RUNG
   RUNG wire#w1
      { S7_Templates := "SrcType := String" } EQ_Contact(in1 := "AutoProcessData".A_Table_2[3].Code, in2 := "ST10_RecipeDB".ParameterElement.A2_TableFixtureCode[3])
      { S7_Templates := "SrcType := String" } NE_Contact(in1 := "AutoProcessData".A_Table_2[3].Code, in2 := '')
      wire#w4
      Move(in := 1, out1 => "AutoProcessData".A_Table_2[3].PartStatus)
   END_RUNG
   RUNG wire#w4
      Not()
      Move(in := 2, out1 => "AutoProcessData".A_Table_2[3].PartStatus)
   END_RUNG
   RUNG wire#w1
      { S7_Templates := "SrcType := String" } EQ_Contact(in1 := "AutoProcessData".A_Table_2[4].Code, in2 := "ST10_RecipeDB".ParameterElement.A2_TableFixtureCode[4])
      { S7_Templates := "SrcType := String" } NE_Contact(in1 := "AutoProcessData".A_Table_2[4].Code, in2 := '')
      wire#w5
      Move(in := 1, out1 => "AutoProcessData".A_Table_2[4].PartStatus)
   END_RUNG
   RUNG wire#w5
      Not()
      Move(in := 2, out1 => "AutoProcessData".A_Table_2[4].PartStatus)
   END_RUNG
   RUNG wire#w1
      { S7_Templates := "SrcType := String" } EQ_Contact(in1 := "AutoProcessData".A_Table_2[5].Code, in2 := "ST10_RecipeDB".ParameterElement.A2_TableFixtureCode[5])
      { S7_Templates := "SrcType := String" } NE_Contact(in1 := "AutoProcessData".A_Table_2[5].Code, in2 := '')
      wire#w6
      Move(in := 1, out1 => "AutoProcessData".A_Table_2[5].PartStatus)
   END_RUNG
   RUNG wire#w6
      Not()
      Move(in := 2, out1 => "AutoProcessData".A_Table_2[5].PartStatus)
   END_RUNG
   RUNG wire#w1
      { S7_Templates := "SrcType := String" } EQ_Contact(in1 := "AutoProcessData".A_Table_2[6].Code, in2 := "ST10_RecipeDB".ParameterElement.A2_TableFixtureCode[6])
      { S7_Templates := "SrcType := String" } NE_Contact(in1 := "AutoProcessData".A_Table_2[6].Code, in2 := '')
      wire#w7
      Move(in := 1, out1 => "AutoProcessData".A_Table_2[6].PartStatus)
   END_RUNG
   RUNG wire#w7
      Not()
      Move(in := 2, out1 => "AutoProcessData".A_Table_2[6].PartStatus)
   END_RUNG
   RUNG wire#w1
      { S7_Templates := "SrcType := String" } EQ_Contact(in1 := "AutoProcessData".A_Table_2[7].Code, in2 := "ST10_RecipeDB".ParameterElement.A2_TableFixtureCode[7])
      { S7_Templates := "SrcType := String" } NE_Contact(in1 := "AutoProcessData".A_Table_2[7].Code, in2 := '')
      wire#w8
      Move(in := 1, out1 => "AutoProcessData".A_Table_2[7].PartStatus)
   END_RUNG
   RUNG wire#w8
      Not()
      Move(in := 2, out1 => "AutoProcessData".A_Table_2[7].PartStatus)
   END_RUNG
   RUNG wire#w1
      { S7_Templates := "SrcType := String" } EQ_Contact(in1 := "AutoProcessData".A_Table_2[8].Code, in2 := "ST10_RecipeDB".ParameterElement.A2_TableFixtureCode[8])
      { S7_Templates := "SrcType := String" } NE_Contact(in1 := "AutoProcessData".A_Table_2[8].Code, in2 := '')
      wire#w9
      Move(in := 1, out1 => "AutoProcessData".A_Table_2[8].PartStatus)
   END_RUNG
   RUNG wire#w9
      Not()
      Move(in := 2, out1 => "AutoProcessData".A_Table_2[8].PartStatus)
   END_RUNG
   RUNG wire#w1
      { S7_Templates := "SrcType := Int" } EQ_Contact(in1 := "AutoProcessData".A_Table_2[1].PartStatus, in2 := 1)
      { S7_Templates := "SrcType := Int" } EQ_Contact(in1 := "AutoProcessData".A_Table_2[2].PartStatus, in2 := 1)
      { S7_Templates := "SrcType := Int" } EQ_Contact(in1 := "AutoProcessData".A_Table_2[3].PartStatus, in2 := 1)
      { S7_Templates := "SrcType := Int" } EQ_Contact(in1 := "AutoProcessData".A_Table_2[4].PartStatus, in2 := 1)
      { S7_Templates := "SrcType := Int" } EQ_Contact(in1 := "AutoProcessData".A_Table_2[5].PartStatus, in2 := 1)
      { S7_Templates := "SrcType := Int" } EQ_Contact(in1 := "AutoProcessData".A_Table_2[6].PartStatus, in2 := 1)
      { S7_Templates := "SrcType := Int" } EQ_Contact(in1 := "AutoProcessData".A_Table_2[7].PartStatus, in2 := 1)
      { S7_Templates := "SrcType := Int" } EQ_Contact(in1 := "AutoProcessData".A_Table_2[8].PartStatus, in2 := 1)
      wire#w10
      Coil( "AutoProcessData".GlobalData.Table2CodeOKFlag )
   END_RUNG
   RUNG wire#w1
      Contact( "ST10_GeneralData".FunctionDeSelect.Global.DeSelectPB_ScanFixture )
   END_RUNG wire#w10
   // the same network as SCL:
   #_w1 := "AlwaysTRUE" AND ("AutoProcessData".A_Table_2[1].Code = "ST10_RecipeDB".ParameterElement.A2_TableFixtureCode[1]) AND ("AutoProcessData".A_Table_2[1].Code <> '');
   IF #_w1 THEN "AutoProcessData".A_Table_2[1].PartStatus := 1; END_IF;
   IF NOT #_w1 THEN "AutoProcessData".A_Table_2[1].PartStatus := 2; END_IF;
   #_w2 := "AlwaysTRUE" AND ("AutoProcessData".A_Table_2[2].Code = "ST10_RecipeDB".ParameterElement.A2_TableFixtureCode[2]) AND ("AutoProcessData".A_Table_2[2].Code <> '');
   IF #_w2 THEN "AutoProcessData".A_Table_2[2].PartStatus := 1; END_IF;
   IF NOT #_w2 THEN "AutoProcessData".A_Table_2[2].PartStatus := 2; END_IF;
   #_w3 := "AlwaysTRUE" AND ("AutoProcessData".A_Table_2[3].Code = "ST10_RecipeDB".ParameterElement.A2_TableFixtureCode[3]) AND ("AutoProcessData".A_Table_2[3].Code <> '');
   IF #_w3 THEN "AutoProcessData".A_Table_2[3].PartStatus := 1; END_IF;
   IF NOT #_w3 THEN "AutoProcessData".A_Table_2[3].PartStatus := 2; END_IF;
   #_w4 := "AlwaysTRUE" AND ("AutoProcessData".A_Table_2[4].Code = "ST10_RecipeDB".ParameterElement.A2_TableFixtureCode[4]) AND ("AutoProcessData".A_Table_2[4].Code <> '');
   IF #_w4 THEN "AutoProcessData".A_Table_2[4].PartStatus := 1; END_IF;
   IF NOT #_w4 THEN "AutoProcessData".A_Table_2[4].PartStatus := 2; END_IF;
   #_w5 := "AlwaysTRUE" AND ("AutoProcessData".A_Table_2[5].Code = "ST10_RecipeDB".ParameterElement.A2_TableFixtureCode[5]) AND ("AutoProcessData".A_Table_2[5].Code <> '');
   IF #_w5 THEN "AutoProcessData".A_Table_2[5].PartStatus := 1; END_IF;
   IF NOT #_w5 THEN "AutoProcessData".A_Table_2[5].PartStatus := 2; END_IF;
   #_w6 := "AlwaysTRUE" AND ("AutoProcessData".A_Table_2[6].Code = "ST10_RecipeDB".ParameterElement.A2_TableFixtureCode[6]) AND ("AutoProcessData".A_Table_2[6].Code <> '');
   IF #_w6 THEN "AutoProcessData".A_Table_2[6].PartStatus := 1; END_IF;
   IF NOT #_w6 THEN "AutoProcessData".A_Table_2[6].PartStatus := 2; END_IF;
   #_w7 := "AlwaysTRUE" AND ("AutoProcessData".A_Table_2[7].Code = "ST10_RecipeDB".ParameterElement.A2_TableFixtureCode[7]) AND ("AutoProcessData".A_Table_2[7].Code <> '');
   IF #_w7 THEN "AutoProcessData".A_Table_2[7].PartStatus := 1; END_IF;
   IF NOT #_w7 THEN "AutoProcessData".A_Table_2[7].PartStatus := 2; END_IF;
   #_w8 := "AlwaysTRUE" AND ("AutoProcessData".A_Table_2[8].Code = "ST10_RecipeDB".ParameterElement.A2_TableFixtureCode[8]) AND ("AutoProcessData".A_Table_2[8].Code <> '');
   IF #_w8 THEN "AutoProcessData".A_Table_2[8].PartStatus := 1; END_IF;
   IF NOT #_w8 THEN "AutoProcessData".A_Table_2[8].PartStatus := 2; END_IF;
   "AutoProcessData".GlobalData.Table2CodeOKFlag := "AlwaysTRUE" AND ((("AutoProcessData".A_Table_2[1].PartStatus = 1) AND ("AutoProcessData".A_Table_2[2].PartStatus = 1) AND ("AutoProcessData".A_Table_2[3].PartStatus = 1) AND ("AutoProcessData".A_Table_2[4].PartStatus = 1) AND ("AutoProcessData".A_Table_2[5].PartStatus = 1) AND ("AutoProcessData".A_Table_2[6].PartStatus = 1) AND ("AutoProcessData".A_Table_2[7].PartStatus = 1) AND ("AutoProcessData".A_Table_2[8].PartStatus = 1)) OR "ST10_GeneralData".FunctionDeSelect.Global.DeSelectPB_ScanFixture);
END_REGION

REGION Network 18: Robot1Grip Code
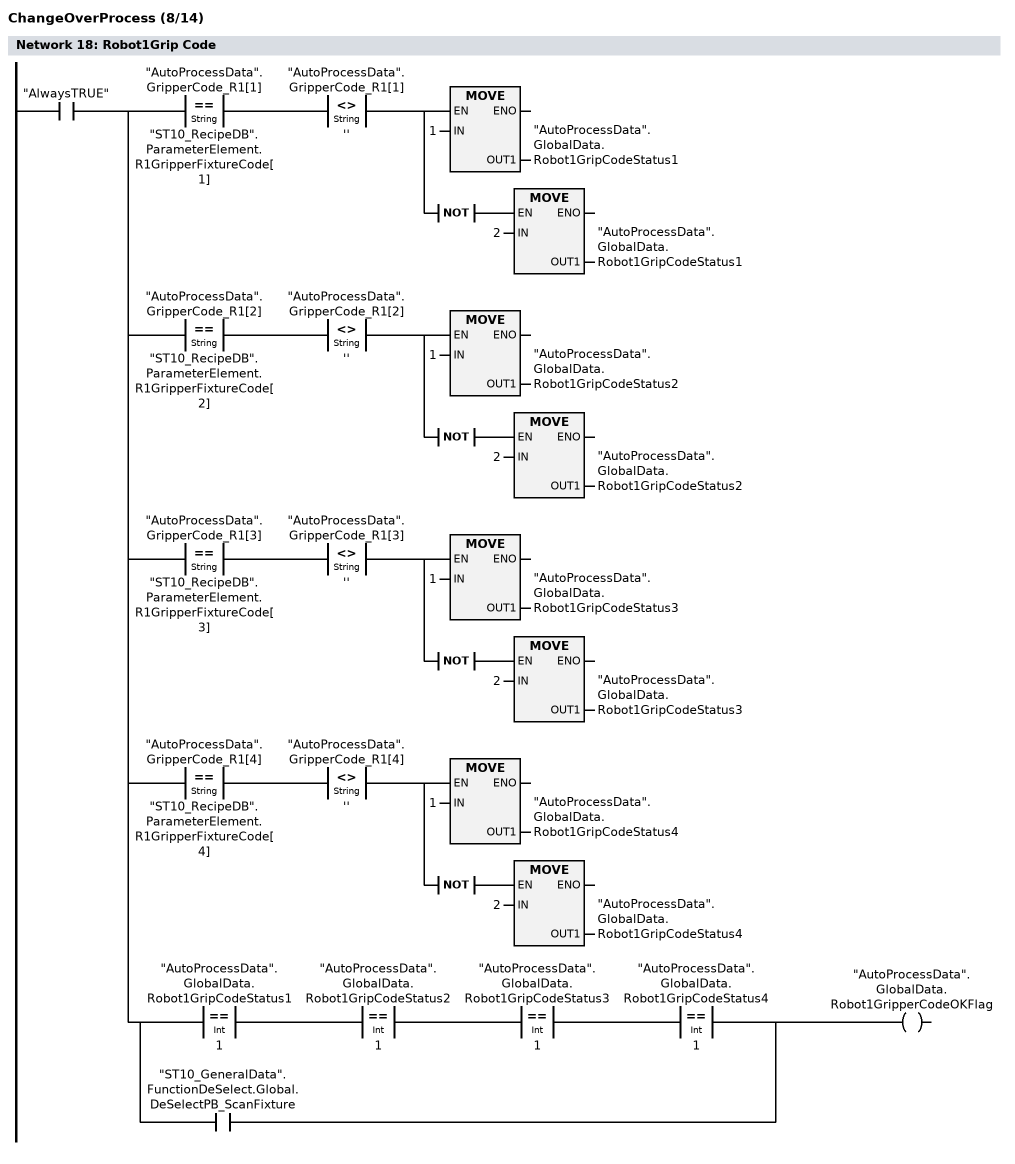
   RUNG wire#powerrail
      Contact( "AlwaysTRUE" )
      wire#w1
      { S7_Templates := "SrcType := String" } EQ_Contact(in1 := "AutoProcessData".GripperCode_R1[1], in2 := "ST10_RecipeDB".ParameterElement.R1GripperFixtureCode[1])
      { S7_Templates := "SrcType := String" } NE_Contact(in1 := "AutoProcessData".GripperCode_R1[1], in2 := '')
      wire#w2
      Move(in := 1, out1 => "AutoProcessData".GlobalData.Robot1GripCodeStatus1)
   END_RUNG
   RUNG wire#w2
      Not()
      Move(in := 2, out1 => "AutoProcessData".GlobalData.Robot1GripCodeStatus1)
   END_RUNG
   RUNG wire#w1
      { S7_Templates := "SrcType := String" } EQ_Contact(in1 := "AutoProcessData".GripperCode_R1[2], in2 := "ST10_RecipeDB".ParameterElement.R1GripperFixtureCode[2])
      { S7_Templates := "SrcType := String" } NE_Contact(in1 := "AutoProcessData".GripperCode_R1[2], in2 := '')
      wire#w3
      Move(in := 1, out1 => "AutoProcessData".GlobalData.Robot1GripCodeStatus2)
   END_RUNG
   RUNG wire#w3
      Not()
      Move(in := 2, out1 => "AutoProcessData".GlobalData.Robot1GripCodeStatus2)
   END_RUNG
   RUNG wire#w1
      { S7_Templates := "SrcType := String" } EQ_Contact(in1 := "AutoProcessData".GripperCode_R1[3], in2 := "ST10_RecipeDB".ParameterElement.R1GripperFixtureCode[3])
      { S7_Templates := "SrcType := String" } NE_Contact(in1 := "AutoProcessData".GripperCode_R1[3], in2 := '')
      wire#w4
      Move(in := 1, out1 => "AutoProcessData".GlobalData.Robot1GripCodeStatus3)
   END_RUNG
   RUNG wire#w4
      Not()
      Move(in := 2, out1 => "AutoProcessData".GlobalData.Robot1GripCodeStatus3)
   END_RUNG
   RUNG wire#w1
      { S7_Templates := "SrcType := String" } EQ_Contact(in1 := "AutoProcessData".GripperCode_R1[4], in2 := "ST10_RecipeDB".ParameterElement.R1GripperFixtureCode[4])
      { S7_Templates := "SrcType := String" } NE_Contact(in1 := "AutoProcessData".GripperCode_R1[4], in2 := '')
      wire#w5
      Move(in := 1, out1 => "AutoProcessData".GlobalData.Robot1GripCodeStatus4)
   END_RUNG
   RUNG wire#w5
      Not()
      Move(in := 2, out1 => "AutoProcessData".GlobalData.Robot1GripCodeStatus4)
   END_RUNG
   RUNG wire#w1
      { S7_Templates := "SrcType := Int" } EQ_Contact(in1 := "AutoProcessData".GlobalData.Robot1GripCodeStatus1, in2 := 1)
      { S7_Templates := "SrcType := Int" } EQ_Contact(in1 := "AutoProcessData".GlobalData.Robot1GripCodeStatus2, in2 := 1)
      { S7_Templates := "SrcType := Int" } EQ_Contact(in1 := "AutoProcessData".GlobalData.Robot1GripCodeStatus3, in2 := 1)
      { S7_Templates := "SrcType := Int" } EQ_Contact(in1 := "AutoProcessData".GlobalData.Robot1GripCodeStatus4, in2 := 1)
      wire#w6
      Coil( "AutoProcessData".GlobalData.Robot1GripperCodeOKFlag )
   END_RUNG
   RUNG wire#w1
      Contact( "ST10_GeneralData".FunctionDeSelect.Global.DeSelectPB_ScanFixture )
   END_RUNG wire#w6
   // the same network as SCL:
   #_w1 := "AlwaysTRUE" AND ("AutoProcessData".GripperCode_R1[1] = "ST10_RecipeDB".ParameterElement.R1GripperFixtureCode[1]) AND ("AutoProcessData".GripperCode_R1[1] <> '');
   IF #_w1 THEN "AutoProcessData".GlobalData.Robot1GripCodeStatus1 := 1; END_IF;
   IF NOT #_w1 THEN "AutoProcessData".GlobalData.Robot1GripCodeStatus1 := 2; END_IF;
   #_w2 := "AlwaysTRUE" AND ("AutoProcessData".GripperCode_R1[2] = "ST10_RecipeDB".ParameterElement.R1GripperFixtureCode[2]) AND ("AutoProcessData".GripperCode_R1[2] <> '');
   IF #_w2 THEN "AutoProcessData".GlobalData.Robot1GripCodeStatus2 := 1; END_IF;
   IF NOT #_w2 THEN "AutoProcessData".GlobalData.Robot1GripCodeStatus2 := 2; END_IF;
   #_w3 := "AlwaysTRUE" AND ("AutoProcessData".GripperCode_R1[3] = "ST10_RecipeDB".ParameterElement.R1GripperFixtureCode[3]) AND ("AutoProcessData".GripperCode_R1[3] <> '');
   IF #_w3 THEN "AutoProcessData".GlobalData.Robot1GripCodeStatus3 := 1; END_IF;
   IF NOT #_w3 THEN "AutoProcessData".GlobalData.Robot1GripCodeStatus3 := 2; END_IF;
   #_w4 := "AlwaysTRUE" AND ("AutoProcessData".GripperCode_R1[4] = "ST10_RecipeDB".ParameterElement.R1GripperFixtureCode[4]) AND ("AutoProcessData".GripperCode_R1[4] <> '');
   IF #_w4 THEN "AutoProcessData".GlobalData.Robot1GripCodeStatus4 := 1; END_IF;
   IF NOT #_w4 THEN "AutoProcessData".GlobalData.Robot1GripCodeStatus4 := 2; END_IF;
   "AutoProcessData".GlobalData.Robot1GripperCodeOKFlag := "AlwaysTRUE" AND ((("AutoProcessData".GlobalData.Robot1GripCodeStatus1 = 1) AND ("AutoProcessData".GlobalData.Robot1GripCodeStatus2 = 1) AND ("AutoProcessData".GlobalData.Robot1GripCodeStatus3 = 1) AND ("AutoProcessData".GlobalData.Robot1GripCodeStatus4 = 1)) OR "ST10_GeneralData".FunctionDeSelect.Global.DeSelectPB_ScanFixture);
END_REGION

REGION Network 19: Robot2Grip Code
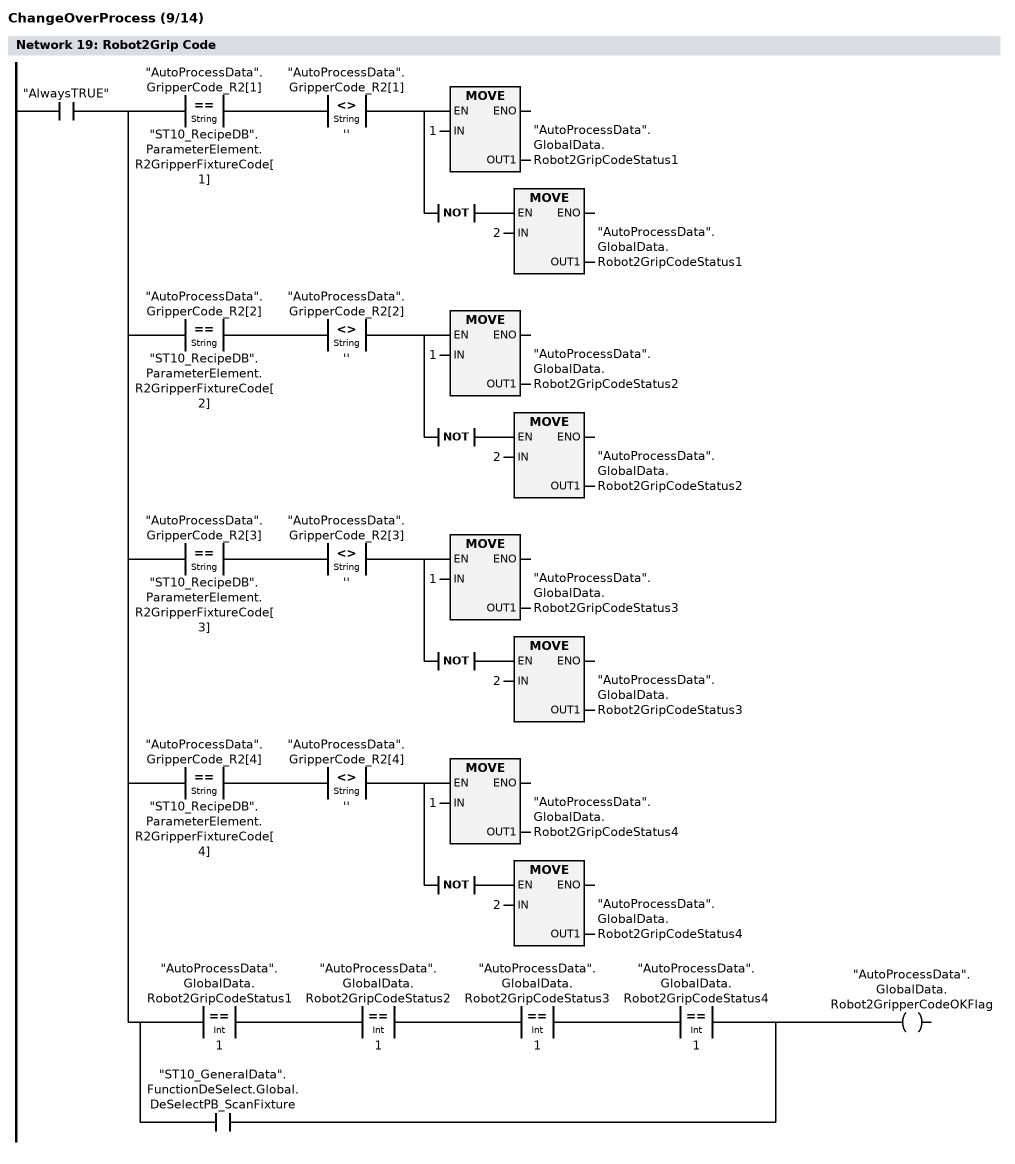
   RUNG wire#powerrail
      Contact( "AlwaysTRUE" )
      wire#w1
      { S7_Templates := "SrcType := String" } EQ_Contact(in1 := "AutoProcessData".GripperCode_R2[1], in2 := "ST10_RecipeDB".ParameterElement.R2GripperFixtureCode[1])
      { S7_Templates := "SrcType := String" } NE_Contact(in1 := "AutoProcessData".GripperCode_R2[1], in2 := '')
      wire#w2
      Move(in := 1, out1 => "AutoProcessData".GlobalData.Robot2GripCodeStatus1)
   END_RUNG
   RUNG wire#w2
      Not()
      Move(in := 2, out1 => "AutoProcessData".GlobalData.Robot2GripCodeStatus1)
   END_RUNG
   RUNG wire#w1
      { S7_Templates := "SrcType := String" } EQ_Contact(in1 := "AutoProcessData".GripperCode_R2[2], in2 := "ST10_RecipeDB".ParameterElement.R2GripperFixtureCode[2])
      { S7_Templates := "SrcType := String" } NE_Contact(in1 := "AutoProcessData".GripperCode_R2[2], in2 := '')
      wire#w3
      Move(in := 1, out1 => "AutoProcessData".GlobalData.Robot2GripCodeStatus2)
   END_RUNG
   RUNG wire#w3
      Not()
      Move(in := 2, out1 => "AutoProcessData".GlobalData.Robot2GripCodeStatus2)
   END_RUNG
   RUNG wire#w1
      { S7_Templates := "SrcType := String" } EQ_Contact(in1 := "AutoProcessData".GripperCode_R2[3], in2 := "ST10_RecipeDB".ParameterElement.R2GripperFixtureCode[3])
      { S7_Templates := "SrcType := String" } NE_Contact(in1 := "AutoProcessData".GripperCode_R2[3], in2 := '')
      wire#w4
      Move(in := 1, out1 => "AutoProcessData".GlobalData.Robot2GripCodeStatus3)
   END_RUNG
   RUNG wire#w4
      Not()
      Move(in := 2, out1 => "AutoProcessData".GlobalData.Robot2GripCodeStatus3)
   END_RUNG
   RUNG wire#w1
      { S7_Templates := "SrcType := String" } EQ_Contact(in1 := "AutoProcessData".GripperCode_R2[4], in2 := "ST10_RecipeDB".ParameterElement.R2GripperFixtureCode[4])
      { S7_Templates := "SrcType := String" } NE_Contact(in1 := "AutoProcessData".GripperCode_R2[4], in2 := '')
      wire#w5
      Move(in := 1, out1 => "AutoProcessData".GlobalData.Robot2GripCodeStatus4)
   END_RUNG
   RUNG wire#w5
      Not()
      Move(in := 2, out1 => "AutoProcessData".GlobalData.Robot2GripCodeStatus4)
   END_RUNG
   RUNG wire#w1
      { S7_Templates := "SrcType := Int" } EQ_Contact(in1 := "AutoProcessData".GlobalData.Robot2GripCodeStatus1, in2 := 1)
      { S7_Templates := "SrcType := Int" } EQ_Contact(in1 := "AutoProcessData".GlobalData.Robot2GripCodeStatus2, in2 := 1)
      { S7_Templates := "SrcType := Int" } EQ_Contact(in1 := "AutoProcessData".GlobalData.Robot2GripCodeStatus3, in2 := 1)
      { S7_Templates := "SrcType := Int" } EQ_Contact(in1 := "AutoProcessData".GlobalData.Robot2GripCodeStatus4, in2 := 1)
      wire#w6
      Coil( "AutoProcessData".GlobalData.Robot2GripperCodeOKFlag )
   END_RUNG
   RUNG wire#w1
      Contact( "ST10_GeneralData".FunctionDeSelect.Global.DeSelectPB_ScanFixture )
   END_RUNG wire#w6
   // the same network as SCL:
   #_w1 := "AlwaysTRUE" AND ("AutoProcessData".GripperCode_R2[1] = "ST10_RecipeDB".ParameterElement.R2GripperFixtureCode[1]) AND ("AutoProcessData".GripperCode_R2[1] <> '');
   IF #_w1 THEN "AutoProcessData".GlobalData.Robot2GripCodeStatus1 := 1; END_IF;
   IF NOT #_w1 THEN "AutoProcessData".GlobalData.Robot2GripCodeStatus1 := 2; END_IF;
   #_w2 := "AlwaysTRUE" AND ("AutoProcessData".GripperCode_R2[2] = "ST10_RecipeDB".ParameterElement.R2GripperFixtureCode[2]) AND ("AutoProcessData".GripperCode_R2[2] <> '');
   IF #_w2 THEN "AutoProcessData".GlobalData.Robot2GripCodeStatus2 := 1; END_IF;
   IF NOT #_w2 THEN "AutoProcessData".GlobalData.Robot2GripCodeStatus2 := 2; END_IF;
   #_w3 := "AlwaysTRUE" AND ("AutoProcessData".GripperCode_R2[3] = "ST10_RecipeDB".ParameterElement.R2GripperFixtureCode[3]) AND ("AutoProcessData".GripperCode_R2[3] <> '');
   IF #_w3 THEN "AutoProcessData".GlobalData.Robot2GripCodeStatus3 := 1; END_IF;
   IF NOT #_w3 THEN "AutoProcessData".GlobalData.Robot2GripCodeStatus3 := 2; END_IF;
   #_w4 := "AlwaysTRUE" AND ("AutoProcessData".GripperCode_R2[4] = "ST10_RecipeDB".ParameterElement.R2GripperFixtureCode[4]) AND ("AutoProcessData".GripperCode_R2[4] <> '');
   IF #_w4 THEN "AutoProcessData".GlobalData.Robot2GripCodeStatus4 := 1; END_IF;
   IF NOT #_w4 THEN "AutoProcessData".GlobalData.Robot2GripCodeStatus4 := 2; END_IF;
   "AutoProcessData".GlobalData.Robot2GripperCodeOKFlag := "AlwaysTRUE" AND ((("AutoProcessData".GlobalData.Robot2GripCodeStatus1 = 1) AND ("AutoProcessData".GlobalData.Robot2GripCodeStatus2 = 1) AND ("AutoProcessData".GlobalData.Robot2GripCodeStatus3 = 1) AND ("AutoProcessData".GlobalData.Robot2GripCodeStatus4 = 1)) OR "ST10_GeneralData".FunctionDeSelect.Global.DeSelectPB_ScanFixture);
END_REGION

REGION Network 20: Robot3Grip Code
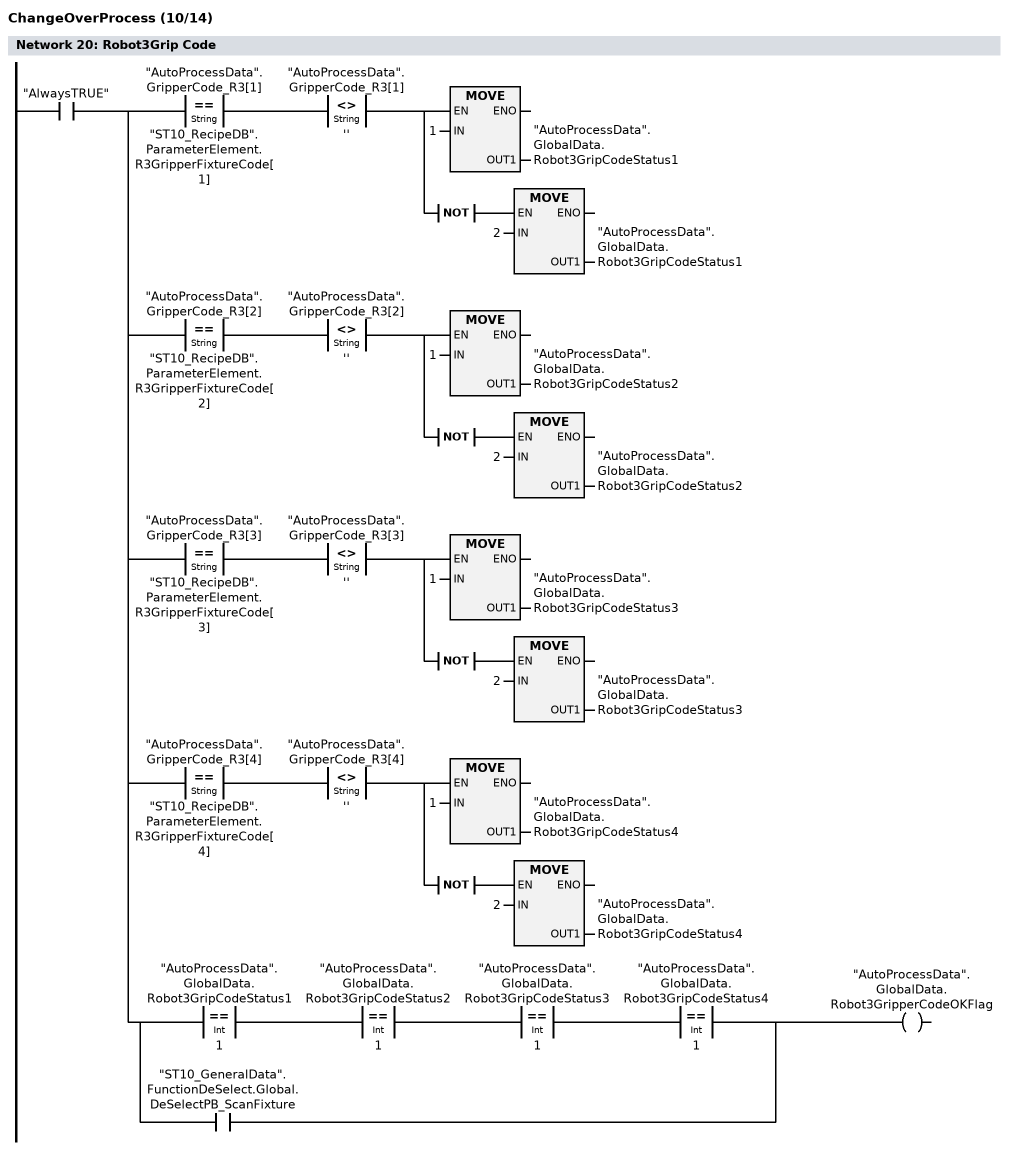
   RUNG wire#powerrail
      Contact( "AlwaysTRUE" )
      wire#w1
      { S7_Templates := "SrcType := String" } EQ_Contact(in1 := "AutoProcessData".GripperCode_R3[1], in2 := "ST10_RecipeDB".ParameterElement.R3GripperFixtureCode[1])
      { S7_Templates := "SrcType := String" } NE_Contact(in1 := "AutoProcessData".GripperCode_R3[1], in2 := '')
      wire#w2
      Move(in := 1, out1 => "AutoProcessData".GlobalData.Robot3GripCodeStatus1)
   END_RUNG
   RUNG wire#w2
      Not()
      Move(in := 2, out1 => "AutoProcessData".GlobalData.Robot3GripCodeStatus1)
   END_RUNG
   RUNG wire#w1
      { S7_Templates := "SrcType := String" } EQ_Contact(in1 := "AutoProcessData".GripperCode_R3[2], in2 := "ST10_RecipeDB".ParameterElement.R3GripperFixtureCode[2])
      { S7_Templates := "SrcType := String" } NE_Contact(in1 := "AutoProcessData".GripperCode_R3[2], in2 := '')
      wire#w3
      Move(in := 1, out1 => "AutoProcessData".GlobalData.Robot3GripCodeStatus2)
   END_RUNG
   RUNG wire#w3
      Not()
      Move(in := 2, out1 => "AutoProcessData".GlobalData.Robot3GripCodeStatus2)
   END_RUNG
   RUNG wire#w1
      { S7_Templates := "SrcType := String" } EQ_Contact(in1 := "AutoProcessData".GripperCode_R3[3], in2 := "ST10_RecipeDB".ParameterElement.R3GripperFixtureCode[3])
      { S7_Templates := "SrcType := String" } NE_Contact(in1 := "AutoProcessData".GripperCode_R3[3], in2 := '')
      wire#w4
      Move(in := 1, out1 => "AutoProcessData".GlobalData.Robot3GripCodeStatus3)
   END_RUNG
   RUNG wire#w4
      Not()
      Move(in := 2, out1 => "AutoProcessData".GlobalData.Robot3GripCodeStatus3)
   END_RUNG
   RUNG wire#w1
      { S7_Templates := "SrcType := String" } EQ_Contact(in1 := "AutoProcessData".GripperCode_R3[4], in2 := "ST10_RecipeDB".ParameterElement.R3GripperFixtureCode[4])
      { S7_Templates := "SrcType := String" } NE_Contact(in1 := "AutoProcessData".GripperCode_R3[4], in2 := '')
      wire#w5
      Move(in := 1, out1 => "AutoProcessData".GlobalData.Robot3GripCodeStatus4)
   END_RUNG
   RUNG wire#w5
      Not()
      Move(in := 2, out1 => "AutoProcessData".GlobalData.Robot3GripCodeStatus4)
   END_RUNG
   RUNG wire#w1
      { S7_Templates := "SrcType := Int" } EQ_Contact(in1 := "AutoProcessData".GlobalData.Robot3GripCodeStatus1, in2 := 1)
      { S7_Templates := "SrcType := Int" } EQ_Contact(in1 := "AutoProcessData".GlobalData.Robot3GripCodeStatus2, in2 := 1)
      { S7_Templates := "SrcType := Int" } EQ_Contact(in1 := "AutoProcessData".GlobalData.Robot3GripCodeStatus3, in2 := 1)
      { S7_Templates := "SrcType := Int" } EQ_Contact(in1 := "AutoProcessData".GlobalData.Robot3GripCodeStatus4, in2 := 1)
      wire#w6
      Coil( "AutoProcessData".GlobalData.Robot3GripperCodeOKFlag )
   END_RUNG
   RUNG wire#w1
      Contact( "ST10_GeneralData".FunctionDeSelect.Global.DeSelectPB_ScanFixture )
   END_RUNG wire#w6
   // the same network as SCL:
   #_w1 := "AlwaysTRUE" AND ("AutoProcessData".GripperCode_R3[1] = "ST10_RecipeDB".ParameterElement.R3GripperFixtureCode[1]) AND ("AutoProcessData".GripperCode_R3[1] <> '');
   IF #_w1 THEN "AutoProcessData".GlobalData.Robot3GripCodeStatus1 := 1; END_IF;
   IF NOT #_w1 THEN "AutoProcessData".GlobalData.Robot3GripCodeStatus1 := 2; END_IF;
   #_w2 := "AlwaysTRUE" AND ("AutoProcessData".GripperCode_R3[2] = "ST10_RecipeDB".ParameterElement.R3GripperFixtureCode[2]) AND ("AutoProcessData".GripperCode_R3[2] <> '');
   IF #_w2 THEN "AutoProcessData".GlobalData.Robot3GripCodeStatus2 := 1; END_IF;
   IF NOT #_w2 THEN "AutoProcessData".GlobalData.Robot3GripCodeStatus2 := 2; END_IF;
   #_w3 := "AlwaysTRUE" AND ("AutoProcessData".GripperCode_R3[3] = "ST10_RecipeDB".ParameterElement.R3GripperFixtureCode[3]) AND ("AutoProcessData".GripperCode_R3[3] <> '');
   IF #_w3 THEN "AutoProcessData".GlobalData.Robot3GripCodeStatus3 := 1; END_IF;
   IF NOT #_w3 THEN "AutoProcessData".GlobalData.Robot3GripCodeStatus3 := 2; END_IF;
   #_w4 := "AlwaysTRUE" AND ("AutoProcessData".GripperCode_R3[4] = "ST10_RecipeDB".ParameterElement.R3GripperFixtureCode[4]) AND ("AutoProcessData".GripperCode_R3[4] <> '');
   IF #_w4 THEN "AutoProcessData".GlobalData.Robot3GripCodeStatus4 := 1; END_IF;
   IF NOT #_w4 THEN "AutoProcessData".GlobalData.Robot3GripCodeStatus4 := 2; END_IF;
   "AutoProcessData".GlobalData.Robot3GripperCodeOKFlag := "AlwaysTRUE" AND ((("AutoProcessData".GlobalData.Robot3GripCodeStatus1 = 1) AND ("AutoProcessData".GlobalData.Robot3GripCodeStatus2 = 1) AND ("AutoProcessData".GlobalData.Robot3GripCodeStatus3 = 1) AND ("AutoProcessData".GlobalData.Robot3GripCodeStatus4 = 1)) OR "ST10_GeneralData".FunctionDeSelect.Global.DeSelectPB_ScanFixture);
END_REGION

REGION Network 21: A1 Fixture Code
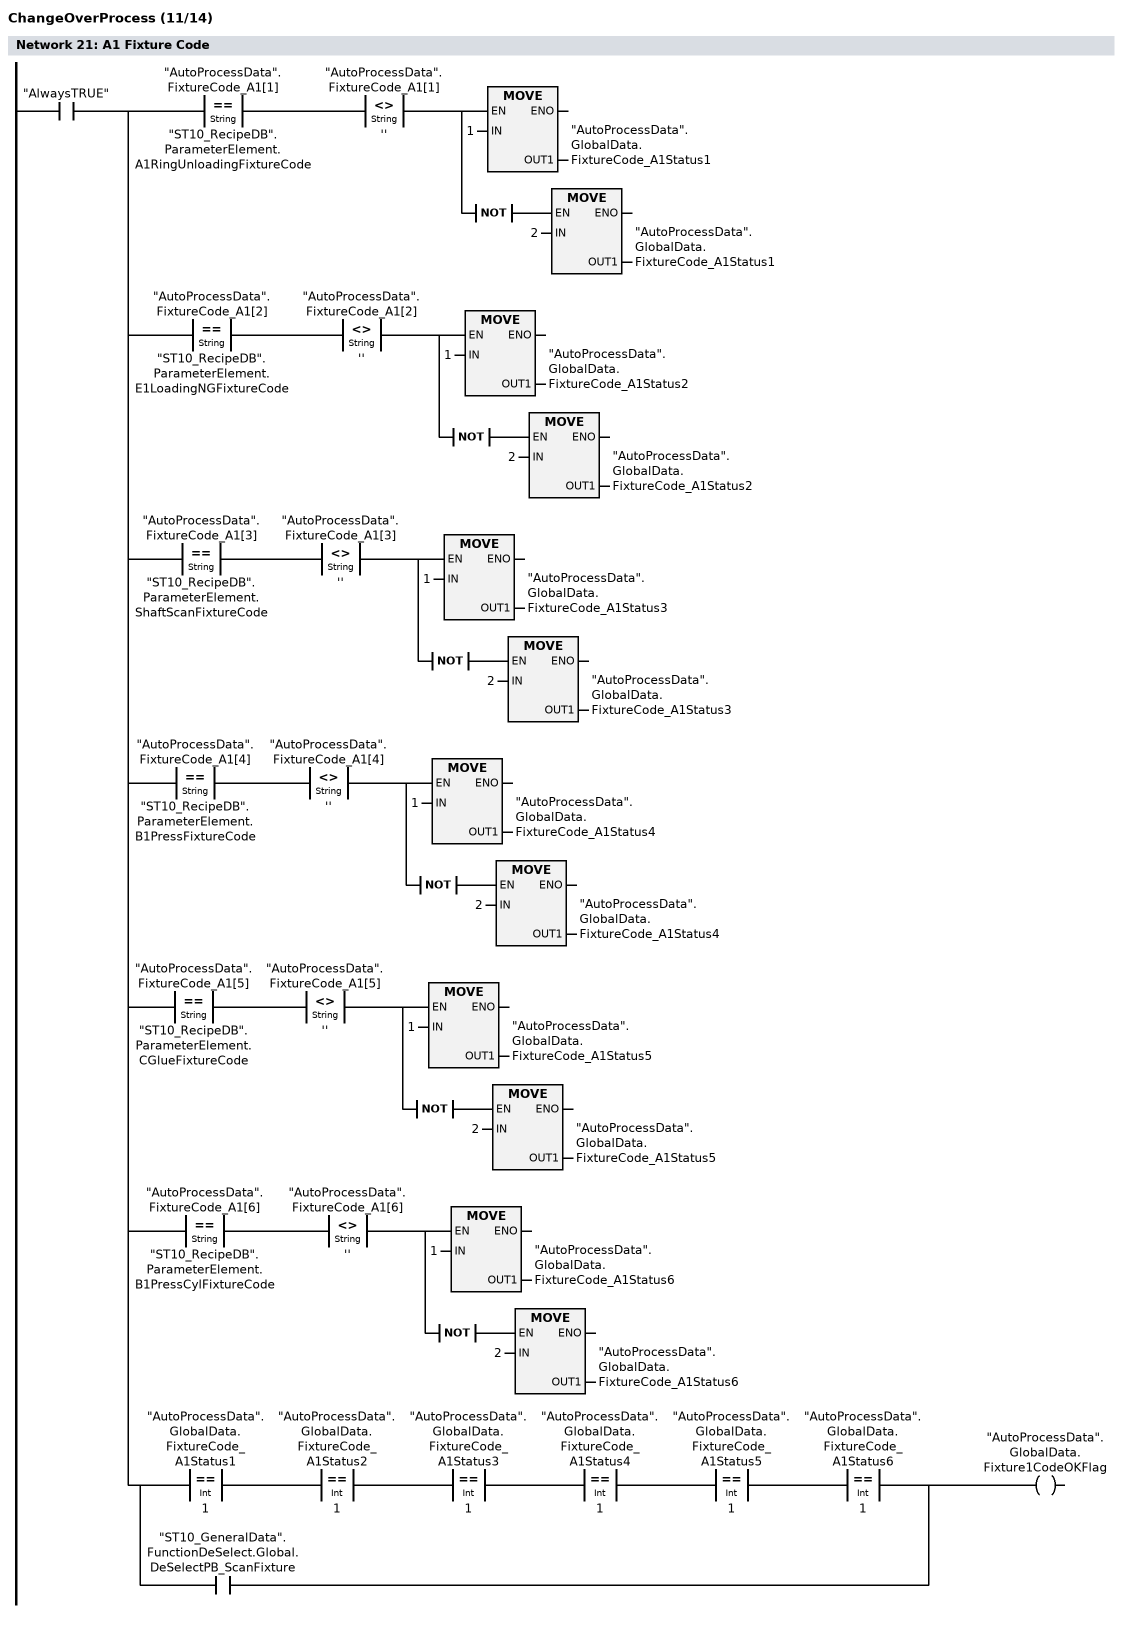
   RUNG wire#powerrail
      Contact( "AlwaysTRUE" )
      wire#w1
      { S7_Templates := "SrcType := String" } EQ_Contact(in1 := "AutoProcessData".FixtureCode_A1[1], in2 := "ST10_RecipeDB".ParameterElement.A1RingUnloadingFixtureCode)
      { S7_Templates := "SrcType := String" } NE_Contact(in1 := "AutoProcessData".FixtureCode_A1[1], in2 := '')
      wire#w2
      Move(in := 1, out1 => "AutoProcessData".GlobalData.FixtureCode_A1Status1)
   END_RUNG
   RUNG wire#w2
      Not()
      Move(in := 2, out1 => "AutoProcessData".GlobalData.FixtureCode_A1Status1)
   END_RUNG
   RUNG wire#w1
      { S7_Templates := "SrcType := String" } EQ_Contact(in1 := "AutoProcessData".FixtureCode_A1[2], in2 := "ST10_RecipeDB".ParameterElement.E1LoadingNGFixtureCode)
      { S7_Templates := "SrcType := String" } NE_Contact(in1 := "AutoProcessData".FixtureCode_A1[2], in2 := '')
      wire#w3
      Move(in := 1, out1 => "AutoProcessData".GlobalData.FixtureCode_A1Status2)
   END_RUNG
   RUNG wire#w3
      Not()
      Move(in := 2, out1 => "AutoProcessData".GlobalData.FixtureCode_A1Status2)
   END_RUNG
   RUNG wire#w1
      { S7_Templates := "SrcType := String" } EQ_Contact(in1 := "AutoProcessData".FixtureCode_A1[3], in2 := "ST10_RecipeDB".ParameterElement.ShaftScanFixtureCode)
      { S7_Templates := "SrcType := String" } NE_Contact(in1 := "AutoProcessData".FixtureCode_A1[3], in2 := '')
      wire#w4
      Move(in := 1, out1 => "AutoProcessData".GlobalData.FixtureCode_A1Status3)
   END_RUNG
   RUNG wire#w4
      Not()
      Move(in := 2, out1 => "AutoProcessData".GlobalData.FixtureCode_A1Status3)
   END_RUNG
   RUNG wire#w1
      { S7_Templates := "SrcType := String" } EQ_Contact(in1 := "AutoProcessData".FixtureCode_A1[4], in2 := "ST10_RecipeDB".ParameterElement.B1PressFixtureCode)
      { S7_Templates := "SrcType := String" } NE_Contact(in1 := "AutoProcessData".FixtureCode_A1[4], in2 := '')
      wire#w5
      Move(in := 1, out1 => "AutoProcessData".GlobalData.FixtureCode_A1Status4)
   END_RUNG
   RUNG wire#w5
      Not()
      Move(in := 2, out1 => "AutoProcessData".GlobalData.FixtureCode_A1Status4)
   END_RUNG
   RUNG wire#w1
      { S7_Templates := "SrcType := String" } EQ_Contact(in1 := "AutoProcessData".FixtureCode_A1[5], in2 := "ST10_RecipeDB".ParameterElement.CGlueFixtureCode)
      { S7_Templates := "SrcType := String" } NE_Contact(in1 := "AutoProcessData".FixtureCode_A1[5], in2 := '')
      wire#w6
      Move(in := 1, out1 => "AutoProcessData".GlobalData.FixtureCode_A1Status5)
   END_RUNG
   RUNG wire#w6
      Not()
      Move(in := 2, out1 => "AutoProcessData".GlobalData.FixtureCode_A1Status5)
   END_RUNG
   RUNG wire#w1
      { S7_Templates := "SrcType := String" } EQ_Contact(in1 := "AutoProcessData".FixtureCode_A1[6], in2 := "ST10_RecipeDB".ParameterElement.B1PressCylFixtureCode)
      { S7_Templates := "SrcType := String" } NE_Contact(in1 := "AutoProcessData".FixtureCode_A1[6], in2 := '')
      wire#w7
      Move(in := 1, out1 => "AutoProcessData".GlobalData.FixtureCode_A1Status6)
   END_RUNG
   RUNG wire#w7
      Not()
      Move(in := 2, out1 => "AutoProcessData".GlobalData.FixtureCode_A1Status6)
   END_RUNG
   RUNG wire#w1
      { S7_Templates := "SrcType := Int" } EQ_Contact(in1 := "AutoProcessData".GlobalData.FixtureCode_A1Status1, in2 := 1)
      { S7_Templates := "SrcType := Int" } EQ_Contact(in1 := "AutoProcessData".GlobalData.FixtureCode_A1Status2, in2 := 1)
      { S7_Templates := "SrcType := Int" } EQ_Contact(in1 := "AutoProcessData".GlobalData.FixtureCode_A1Status3, in2 := 1)
      { S7_Templates := "SrcType := Int" } EQ_Contact(in1 := "AutoProcessData".GlobalData.FixtureCode_A1Status4, in2 := 1)
      { S7_Templates := "SrcType := Int" } EQ_Contact(in1 := "AutoProcessData".GlobalData.FixtureCode_A1Status5, in2 := 1)
      { S7_Templates := "SrcType := Int" } EQ_Contact(in1 := "AutoProcessData".GlobalData.FixtureCode_A1Status6, in2 := 1)
      wire#w8
      Coil( "AutoProcessData".GlobalData.Fixture1CodeOKFlag )
   END_RUNG
   RUNG wire#w1
      Contact( "ST10_GeneralData".FunctionDeSelect.Global.DeSelectPB_ScanFixture )
   END_RUNG wire#w8
   // the same network as SCL:
   #_w1 := "AlwaysTRUE" AND ("AutoProcessData".FixtureCode_A1[1] = "ST10_RecipeDB".ParameterElement.A1RingUnloadingFixtureCode) AND ("AutoProcessData".FixtureCode_A1[1] <> '');
   IF #_w1 THEN "AutoProcessData".GlobalData.FixtureCode_A1Status1 := 1; END_IF;
   IF NOT #_w1 THEN "AutoProcessData".GlobalData.FixtureCode_A1Status1 := 2; END_IF;
   #_w2 := "AlwaysTRUE" AND ("AutoProcessData".FixtureCode_A1[2] = "ST10_RecipeDB".ParameterElement.E1LoadingNGFixtureCode) AND ("AutoProcessData".FixtureCode_A1[2] <> '');
   IF #_w2 THEN "AutoProcessData".GlobalData.FixtureCode_A1Status2 := 1; END_IF;
   IF NOT #_w2 THEN "AutoProcessData".GlobalData.FixtureCode_A1Status2 := 2; END_IF;
   #_w3 := "AlwaysTRUE" AND ("AutoProcessData".FixtureCode_A1[3] = "ST10_RecipeDB".ParameterElement.ShaftScanFixtureCode) AND ("AutoProcessData".FixtureCode_A1[3] <> '');
   IF #_w3 THEN "AutoProcessData".GlobalData.FixtureCode_A1Status3 := 1; END_IF;
   IF NOT #_w3 THEN "AutoProcessData".GlobalData.FixtureCode_A1Status3 := 2; END_IF;
   #_w4 := "AlwaysTRUE" AND ("AutoProcessData".FixtureCode_A1[4] = "ST10_RecipeDB".ParameterElement.B1PressFixtureCode) AND ("AutoProcessData".FixtureCode_A1[4] <> '');
   IF #_w4 THEN "AutoProcessData".GlobalData.FixtureCode_A1Status4 := 1; END_IF;
   IF NOT #_w4 THEN "AutoProcessData".GlobalData.FixtureCode_A1Status4 := 2; END_IF;
   #_w5 := "AlwaysTRUE" AND ("AutoProcessData".FixtureCode_A1[5] = "ST10_RecipeDB".ParameterElement.CGlueFixtureCode) AND ("AutoProcessData".FixtureCode_A1[5] <> '');
   IF #_w5 THEN "AutoProcessData".GlobalData.FixtureCode_A1Status5 := 1; END_IF;
   IF NOT #_w5 THEN "AutoProcessData".GlobalData.FixtureCode_A1Status5 := 2; END_IF;
   #_w6 := "AlwaysTRUE" AND ("AutoProcessData".FixtureCode_A1[6] = "ST10_RecipeDB".ParameterElement.B1PressCylFixtureCode) AND ("AutoProcessData".FixtureCode_A1[6] <> '');
   IF #_w6 THEN "AutoProcessData".GlobalData.FixtureCode_A1Status6 := 1; END_IF;
   IF NOT #_w6 THEN "AutoProcessData".GlobalData.FixtureCode_A1Status6 := 2; END_IF;
   "AutoProcessData".GlobalData.Fixture1CodeOKFlag := "AlwaysTRUE" AND ((("AutoProcessData".GlobalData.FixtureCode_A1Status1 = 1) AND ("AutoProcessData".GlobalData.FixtureCode_A1Status2 = 1) AND ("AutoProcessData".GlobalData.FixtureCode_A1Status3 = 1) AND ("AutoProcessData".GlobalData.FixtureCode_A1Status4 = 1) AND ("AutoProcessData".GlobalData.FixtureCode_A1Status5 = 1) AND ("AutoProcessData".GlobalData.FixtureCode_A1Status6 = 1)) OR "ST10_GeneralData".FunctionDeSelect.Global.DeSelectPB_ScanFixture);
END_REGION

REGION Network 22: A2 Fixture Code
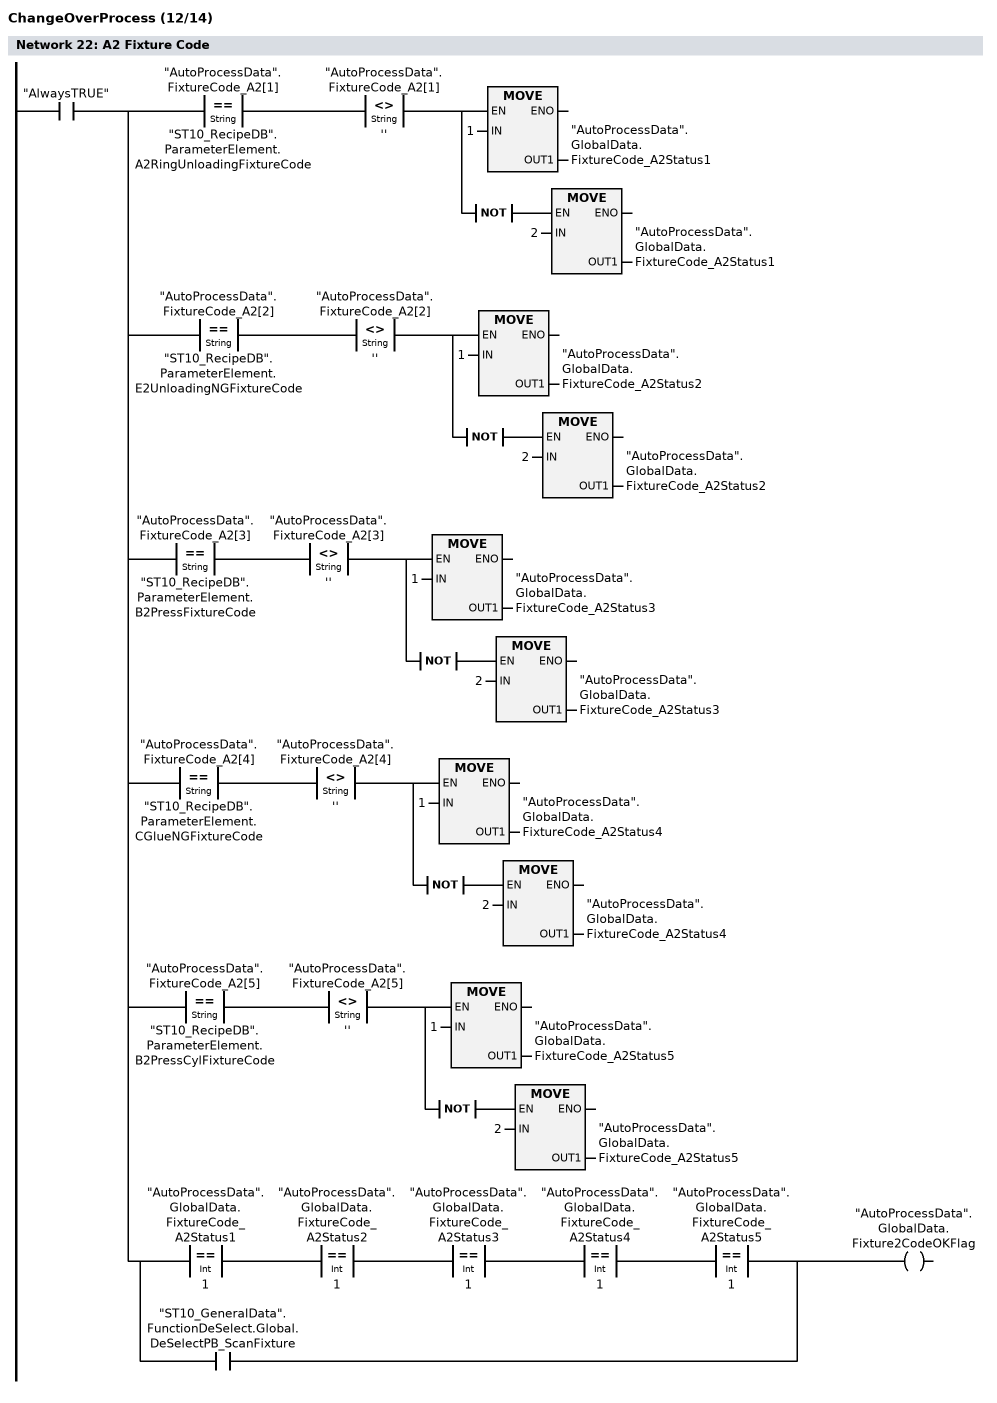
   RUNG wire#powerrail
      Contact( "AlwaysTRUE" )
      wire#w1
      { S7_Templates := "SrcType := String" } EQ_Contact(in1 := "AutoProcessData".FixtureCode_A2[1], in2 := "ST10_RecipeDB".ParameterElement.A2RingUnloadingFixtureCode)
      { S7_Templates := "SrcType := String" } NE_Contact(in1 := "AutoProcessData".FixtureCode_A2[1], in2 := '')
      wire#w2
      Move(in := 1, out1 => "AutoProcessData".GlobalData.FixtureCode_A2Status1)
   END_RUNG
   RUNG wire#w2
      Not()
      Move(in := 2, out1 => "AutoProcessData".GlobalData.FixtureCode_A2Status1)
   END_RUNG
   RUNG wire#w1
      { S7_Templates := "SrcType := String" } EQ_Contact(in1 := "AutoProcessData".FixtureCode_A2[2], in2 := "ST10_RecipeDB".ParameterElement.E2UnloadingNGFixtureCode)
      { S7_Templates := "SrcType := String" } NE_Contact(in1 := "AutoProcessData".FixtureCode_A2[2], in2 := '')
      wire#w3
      Move(in := 1, out1 => "AutoProcessData".GlobalData.FixtureCode_A2Status2)
   END_RUNG
   RUNG wire#w3
      Not()
      Move(in := 2, out1 => "AutoProcessData".GlobalData.FixtureCode_A2Status2)
   END_RUNG
   RUNG wire#w1
      { S7_Templates := "SrcType := String" } EQ_Contact(in1 := "AutoProcessData".FixtureCode_A2[3], in2 := "ST10_RecipeDB".ParameterElement.B2PressFixtureCode)
      { S7_Templates := "SrcType := String" } NE_Contact(in1 := "AutoProcessData".FixtureCode_A2[3], in2 := '')
      wire#w4
      Move(in := 1, out1 => "AutoProcessData".GlobalData.FixtureCode_A2Status3)
   END_RUNG
   RUNG wire#w4
      Not()
      Move(in := 2, out1 => "AutoProcessData".GlobalData.FixtureCode_A2Status3)
   END_RUNG
   RUNG wire#w1
      { S7_Templates := "SrcType := String" } EQ_Contact(in1 := "AutoProcessData".FixtureCode_A2[4], in2 := "ST10_RecipeDB".ParameterElement.CGlueNGFixtureCode)
      { S7_Templates := "SrcType := String" } NE_Contact(in1 := "AutoProcessData".FixtureCode_A2[4], in2 := '')
      wire#w5
      Move(in := 1, out1 => "AutoProcessData".GlobalData.FixtureCode_A2Status4)
   END_RUNG
   RUNG wire#w5
      Not()
      Move(in := 2, out1 => "AutoProcessData".GlobalData.FixtureCode_A2Status4)
   END_RUNG
   RUNG wire#w1
      { S7_Templates := "SrcType := String" } EQ_Contact(in1 := "AutoProcessData".FixtureCode_A2[5], in2 := "ST10_RecipeDB".ParameterElement.B2PressCylFixtureCode)
      { S7_Templates := "SrcType := String" } NE_Contact(in1 := "AutoProcessData".FixtureCode_A2[5], in2 := '')
      wire#w6
      Move(in := 1, out1 => "AutoProcessData".GlobalData.FixtureCode_A2Status5)
   END_RUNG
   RUNG wire#w6
      Not()
      Move(in := 2, out1 => "AutoProcessData".GlobalData.FixtureCode_A2Status5)
   END_RUNG
   RUNG wire#w1
      { S7_Templates := "SrcType := Int" } EQ_Contact(in1 := "AutoProcessData".GlobalData.FixtureCode_A2Status1, in2 := 1)
      { S7_Templates := "SrcType := Int" } EQ_Contact(in1 := "AutoProcessData".GlobalData.FixtureCode_A2Status2, in2 := 1)
      { S7_Templates := "SrcType := Int" } EQ_Contact(in1 := "AutoProcessData".GlobalData.FixtureCode_A2Status3, in2 := 1)
      { S7_Templates := "SrcType := Int" } EQ_Contact(in1 := "AutoProcessData".GlobalData.FixtureCode_A2Status4, in2 := 1)
      { S7_Templates := "SrcType := Int" } EQ_Contact(in1 := "AutoProcessData".GlobalData.FixtureCode_A2Status5, in2 := 1)
      wire#w7
      Coil( "AutoProcessData".GlobalData.Fixture2CodeOKFlag )
   END_RUNG
   RUNG wire#w1
      Contact( "ST10_GeneralData".FunctionDeSelect.Global.DeSelectPB_ScanFixture )
   END_RUNG wire#w7
   // the same network as SCL:
   #_w1 := "AlwaysTRUE" AND ("AutoProcessData".FixtureCode_A2[1] = "ST10_RecipeDB".ParameterElement.A2RingUnloadingFixtureCode) AND ("AutoProcessData".FixtureCode_A2[1] <> '');
   IF #_w1 THEN "AutoProcessData".GlobalData.FixtureCode_A2Status1 := 1; END_IF;
   IF NOT #_w1 THEN "AutoProcessData".GlobalData.FixtureCode_A2Status1 := 2; END_IF;
   #_w2 := "AlwaysTRUE" AND ("AutoProcessData".FixtureCode_A2[2] = "ST10_RecipeDB".ParameterElement.E2UnloadingNGFixtureCode) AND ("AutoProcessData".FixtureCode_A2[2] <> '');
   IF #_w2 THEN "AutoProcessData".GlobalData.FixtureCode_A2Status2 := 1; END_IF;
   IF NOT #_w2 THEN "AutoProcessData".GlobalData.FixtureCode_A2Status2 := 2; END_IF;
   #_w3 := "AlwaysTRUE" AND ("AutoProcessData".FixtureCode_A2[3] = "ST10_RecipeDB".ParameterElement.B2PressFixtureCode) AND ("AutoProcessData".FixtureCode_A2[3] <> '');
   IF #_w3 THEN "AutoProcessData".GlobalData.FixtureCode_A2Status3 := 1; END_IF;
   IF NOT #_w3 THEN "AutoProcessData".GlobalData.FixtureCode_A2Status3 := 2; END_IF;
   #_w4 := "AlwaysTRUE" AND ("AutoProcessData".FixtureCode_A2[4] = "ST10_RecipeDB".ParameterElement.CGlueNGFixtureCode) AND ("AutoProcessData".FixtureCode_A2[4] <> '');
   IF #_w4 THEN "AutoProcessData".GlobalData.FixtureCode_A2Status4 := 1; END_IF;
   IF NOT #_w4 THEN "AutoProcessData".GlobalData.FixtureCode_A2Status4 := 2; END_IF;
   #_w5 := "AlwaysTRUE" AND ("AutoProcessData".FixtureCode_A2[5] = "ST10_RecipeDB".ParameterElement.B2PressCylFixtureCode) AND ("AutoProcessData".FixtureCode_A2[5] <> '');
   IF #_w5 THEN "AutoProcessData".GlobalData.FixtureCode_A2Status5 := 1; END_IF;
   IF NOT #_w5 THEN "AutoProcessData".GlobalData.FixtureCode_A2Status5 := 2; END_IF;
   "AutoProcessData".GlobalData.Fixture2CodeOKFlag := "AlwaysTRUE" AND ((("AutoProcessData".GlobalData.FixtureCode_A2Status1 = 1) AND ("AutoProcessData".GlobalData.FixtureCode_A2Status2 = 1) AND ("AutoProcessData".GlobalData.FixtureCode_A2Status3 = 1) AND ("AutoProcessData".GlobalData.FixtureCode_A2Status4 = 1) AND ("AutoProcessData".GlobalData.FixtureCode_A2Status5 = 1)) OR "ST10_GeneralData".FunctionDeSelect.Global.DeSelectPB_ScanFixture);
END_REGION

REGION Network 23: ChangeOverFinish
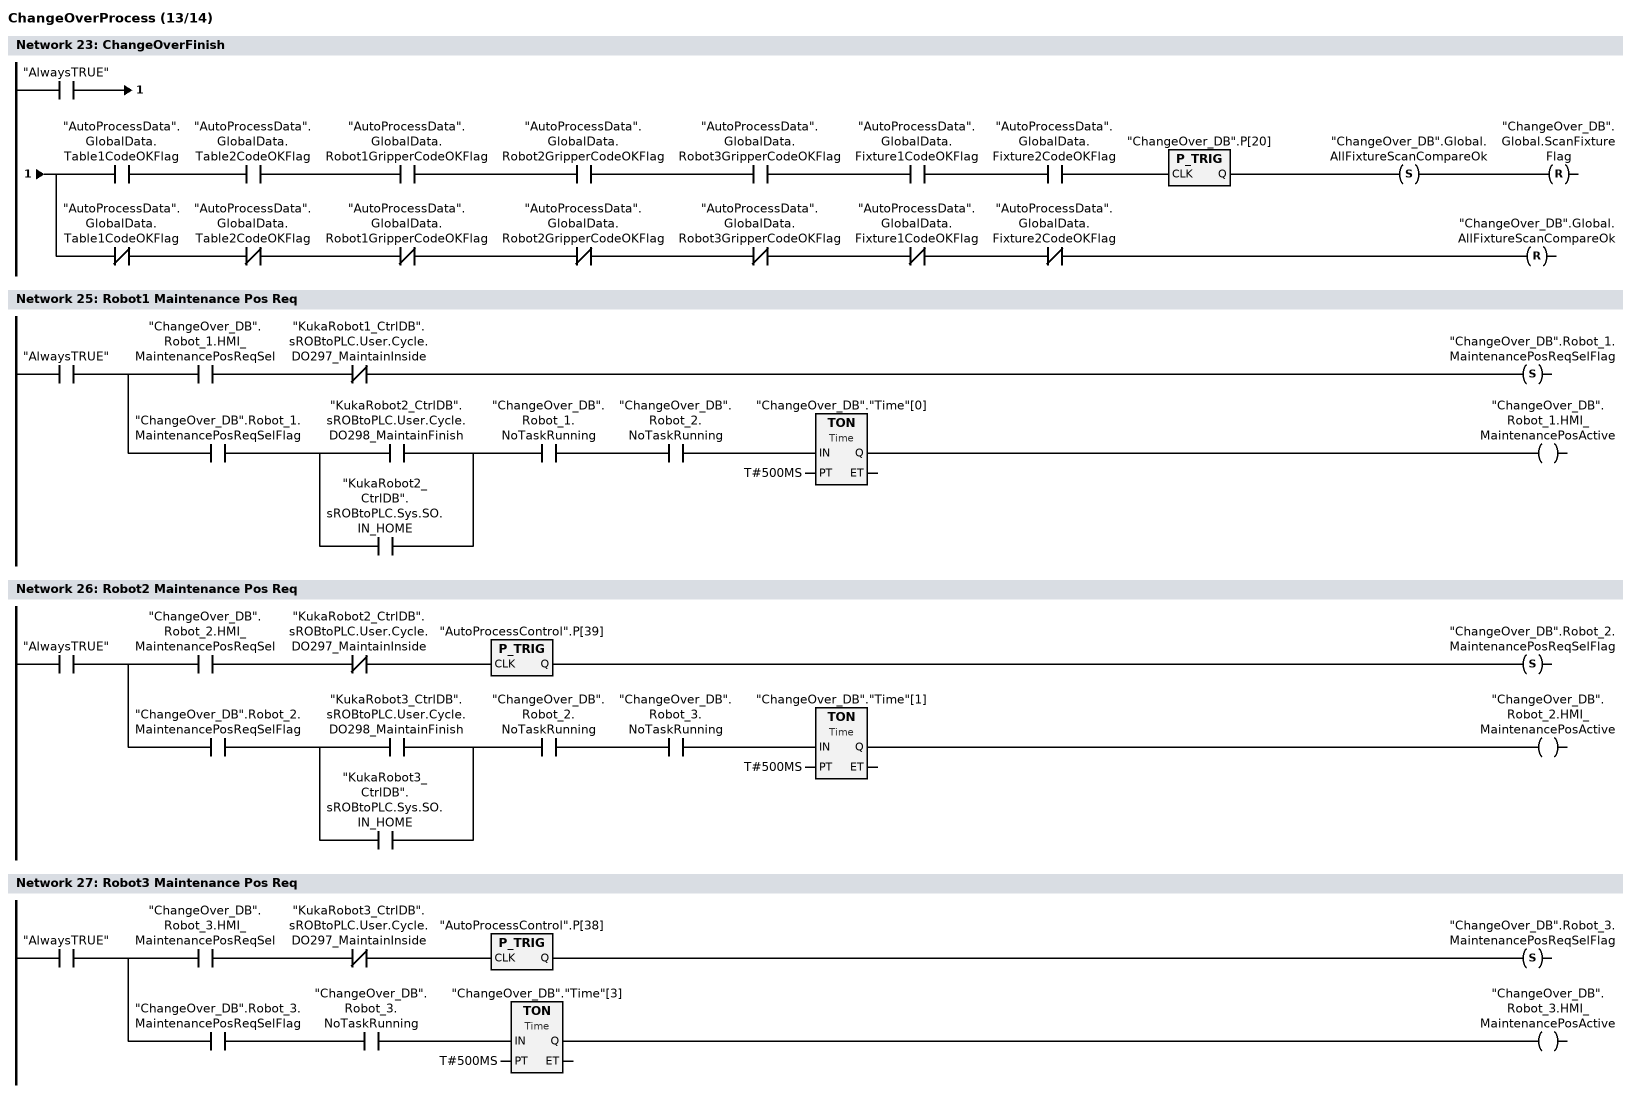
   RUNG wire#powerrail
      Contact( "AlwaysTRUE" )
      wire#w1
      Contact( "AutoProcessData".GlobalData.Table1CodeOKFlag )
      Contact( "AutoProcessData".GlobalData.Table2CodeOKFlag )
      Contact( "AutoProcessData".GlobalData.Robot1GripperCodeOKFlag )
      Contact( "AutoProcessData".GlobalData.Robot2GripperCodeOKFlag )
      Contact( "AutoProcessData".GlobalData.Robot3GripperCodeOKFlag )
      Contact( "AutoProcessData".GlobalData.Fixture1CodeOKFlag )
      Contact( "AutoProcessData".GlobalData.Fixture2CodeOKFlag )
      P_Trig( "ChangeOver_DB".P[20] )
      S_Coil( "ChangeOver_DB".Global.AllFixtureScanCompareOk )
      R_Coil( "ChangeOver_DB".Global.ScanFixtureFlag )
   END_RUNG
   RUNG wire#w1
      I_Contact( "AutoProcessData".GlobalData.Table1CodeOKFlag )
      I_Contact( "AutoProcessData".GlobalData.Table2CodeOKFlag )
      I_Contact( "AutoProcessData".GlobalData.Robot1GripperCodeOKFlag )
      I_Contact( "AutoProcessData".GlobalData.Robot2GripperCodeOKFlag )
      I_Contact( "AutoProcessData".GlobalData.Robot3GripperCodeOKFlag )
      I_Contact( "AutoProcessData".GlobalData.Fixture1CodeOKFlag )
      I_Contact( "AutoProcessData".GlobalData.Fixture2CodeOKFlag )
      R_Coil( "ChangeOver_DB".Global.AllFixtureScanCompareOk )
   END_RUNG
   // the same network as SCL:
   #_w1 := "AlwaysTRUE" AND "AutoProcessData".GlobalData.Table1CodeOKFlag AND "AutoProcessData".GlobalData.Table2CodeOKFlag AND "AutoProcessData".GlobalData.Robot1GripperCodeOKFlag AND "AutoProcessData".GlobalData.Robot2GripperCodeOKFlag AND "AutoProcessData".GlobalData.Robot3GripperCodeOKFlag AND "AutoProcessData".GlobalData.Fixture1CodeOKFlag AND "AutoProcessData".GlobalData.Fixture2CodeOKFlag;
   #_w2 := #_w1 AND NOT "ChangeOver_DB".P[20];   // rising edge
   "ChangeOver_DB".P[20] := #_w1;
   IF #_w2 THEN
       "ChangeOver_DB".Global.AllFixtureScanCompareOk := TRUE;
       "ChangeOver_DB".Global.ScanFixtureFlag := FALSE;
   END_IF;
   IF "AlwaysTRUE" AND NOT "AutoProcessData".GlobalData.Table1CodeOKFlag AND NOT "AutoProcessData".GlobalData.Table2CodeOKFlag AND NOT "AutoProcessData".GlobalData.Robot1GripperCodeOKFlag AND NOT "AutoProcessData".GlobalData.Robot2GripperCodeOKFlag AND NOT "AutoProcessData".GlobalData.Robot3GripperCodeOKFlag AND NOT "AutoProcessData".GlobalData.Fixture1CodeOKFlag AND NOT "AutoProcessData".GlobalData.Fixture2CodeOKFlag THEN
       "ChangeOver_DB".Global.AllFixtureScanCompareOk := FALSE;
   END_IF;
END_REGION

REGION Network 24: ---------------------------------- Manual mode Set maintenance pos / Home pos req ------------------------------------------
END_REGION

REGION Network 25: Robot1 Maintenance Pos Req
   RUNG wire#powerrail
      Contact( "AlwaysTRUE" )
      wire#w1
      Contact( "ChangeOver_DB".Robot_1.HMI_MaintenancePosReqSel )
      I_Contact( "KukaRobot1_CtrlDB".sROBtoPLC.User.Cycle.DO297_MaintainInside )
      S_Coil( "ChangeOver_DB".Robot_1.MaintenancePosReqSelFlag )
   END_RUNG
   RUNG wire#w1
      Contact( "ChangeOver_DB".Robot_1.MaintenancePosReqSelFlag )
      wire#w2
      Contact( "KukaRobot2_CtrlDB".sROBtoPLC.User.Cycle.DO298_MaintainFinish )
      wire#w3
      Contact( "ChangeOver_DB".Robot_1.NoTaskRunning )
      Contact( "ChangeOver_DB".Robot_2.NoTaskRunning )
      { S7_Templates := "time_type := Time" } "ChangeOver_DB"."Time"[0].TON(pt := T#500MS, et =>)
      Coil( "ChangeOver_DB".Robot_1.HMI_MaintenancePosActive )
   END_RUNG
   RUNG wire#w2
      Contact( "KukaRobot2_CtrlDB".sROBtoPLC.Sys.SO.IN_HOME )
   END_RUNG wire#w3
   // the same network as SCL:
   IF "AlwaysTRUE" AND "ChangeOver_DB".Robot_1.HMI_MaintenancePosReqSel AND NOT "KukaRobot1_CtrlDB".sROBtoPLC.User.Cycle.DO297_MaintainInside THEN
       "ChangeOver_DB".Robot_1.MaintenancePosReqSelFlag := TRUE;
   END_IF;
   "ChangeOver_DB"."Time"[0].TON(IN := "AlwaysTRUE" AND "ChangeOver_DB".Robot_1.MaintenancePosReqSelFlag AND ("KukaRobot2_CtrlDB".sROBtoPLC.User.Cycle.DO298_MaintainFinish OR "KukaRobot2_CtrlDB".sROBtoPLC.Sys.SO.IN_HOME) AND "ChangeOver_DB".Robot_1.NoTaskRunning AND "ChangeOver_DB".Robot_2.NoTaskRunning,
                           PT := T#500MS);
   "ChangeOver_DB".Robot_1.HMI_MaintenancePosActive := "ChangeOver_DB"."Time"[0].Q;
END_REGION

REGION Network 26: Robot2 Maintenance Pos Req
   RUNG wire#powerrail
      Contact( "AlwaysTRUE" )
      wire#w1
      Contact( "ChangeOver_DB".Robot_2.HMI_MaintenancePosReqSel )
      I_Contact( "KukaRobot2_CtrlDB".sROBtoPLC.User.Cycle.DO297_MaintainInside )
      P_Trig( "AutoProcessControl".P[39] )
      S_Coil( "ChangeOver_DB".Robot_2.MaintenancePosReqSelFlag )
   END_RUNG
   RUNG wire#w1
      Contact( "ChangeOver_DB".Robot_2.MaintenancePosReqSelFlag )
      wire#w2
      Contact( "KukaRobot3_CtrlDB".sROBtoPLC.User.Cycle.DO298_MaintainFinish )
      wire#w3
      Contact( "ChangeOver_DB".Robot_2.NoTaskRunning )
      Contact( "ChangeOver_DB".Robot_3.NoTaskRunning )
      { S7_Templates := "time_type := Time" } "ChangeOver_DB"."Time"[1].TON(pt := T#500MS, et =>)
      Coil( "ChangeOver_DB".Robot_2.HMI_MaintenancePosActive )
   END_RUNG
   RUNG wire#w2
      Contact( "KukaRobot3_CtrlDB".sROBtoPLC.Sys.SO.IN_HOME )
   END_RUNG wire#w3
   // the same network as SCL:
   #_w1 := "AlwaysTRUE" AND "ChangeOver_DB".Robot_2.HMI_MaintenancePosReqSel AND NOT "KukaRobot2_CtrlDB".sROBtoPLC.User.Cycle.DO297_MaintainInside;
   #_w2 := #_w1 AND NOT "AutoProcessControl".P[39];   // rising edge
   "AutoProcessControl".P[39] := #_w1;
   IF #_w2 THEN "ChangeOver_DB".Robot_2.MaintenancePosReqSelFlag := TRUE; END_IF;
   "ChangeOver_DB"."Time"[1].TON(IN := "AlwaysTRUE" AND "ChangeOver_DB".Robot_2.MaintenancePosReqSelFlag AND ("KukaRobot3_CtrlDB".sROBtoPLC.User.Cycle.DO298_MaintainFinish OR "KukaRobot3_CtrlDB".sROBtoPLC.Sys.SO.IN_HOME) AND "ChangeOver_DB".Robot_2.NoTaskRunning AND "ChangeOver_DB".Robot_3.NoTaskRunning,
                           PT := T#500MS);
   "ChangeOver_DB".Robot_2.HMI_MaintenancePosActive := "ChangeOver_DB"."Time"[1].Q;
END_REGION

REGION Network 27: Robot3 Maintenance Pos Req
   RUNG wire#powerrail
      Contact( "AlwaysTRUE" )
      wire#w1
      Contact( "ChangeOver_DB".Robot_3.HMI_MaintenancePosReqSel )
      I_Contact( "KukaRobot3_CtrlDB".sROBtoPLC.User.Cycle.DO297_MaintainInside )
      P_Trig( "AutoProcessControl".P[38] )
      S_Coil( "ChangeOver_DB".Robot_3.MaintenancePosReqSelFlag )
   END_RUNG
   RUNG wire#w1
      Contact( "ChangeOver_DB".Robot_3.MaintenancePosReqSelFlag )
      Contact( "ChangeOver_DB".Robot_3.NoTaskRunning )
      { S7_Templates := "time_type := Time" } "ChangeOver_DB"."Time"[3].TON(pt := T#500MS, et =>)
      Coil( "ChangeOver_DB".Robot_3.HMI_MaintenancePosActive )
   END_RUNG
   // the same network as SCL:
   #_w1 := "AlwaysTRUE" AND "ChangeOver_DB".Robot_3.HMI_MaintenancePosReqSel AND NOT "KukaRobot3_CtrlDB".sROBtoPLC.User.Cycle.DO297_MaintainInside;
   #_w2 := #_w1 AND NOT "AutoProcessControl".P[38];   // rising edge
   "AutoProcessControl".P[38] := #_w1;
   IF #_w2 THEN "ChangeOver_DB".Robot_3.MaintenancePosReqSelFlag := TRUE; END_IF;
   "ChangeOver_DB"."Time"[3].TON(IN := "AlwaysTRUE" AND "ChangeOver_DB".Robot_3.MaintenancePosReqSelFlag AND "ChangeOver_DB".Robot_3.NoTaskRunning,
                           PT := T#500MS);
   "ChangeOver_DB".Robot_3.HMI_MaintenancePosActive := "ChangeOver_DB"."Time"[3].Q;
END_REGION

REGION Network 28: Station empty
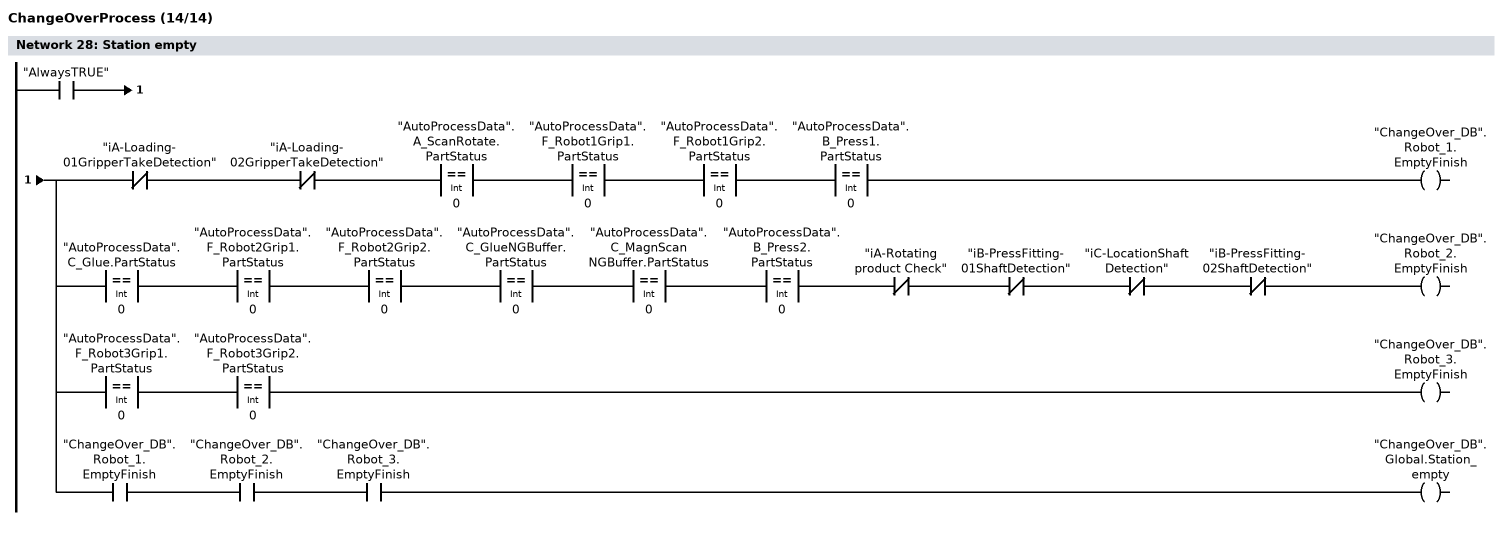
   RUNG wire#powerrail
      Contact( "AlwaysTRUE" )
      wire#w1
      I_Contact( "iA-Loading-01GripperTakeDetection" )
      I_Contact( "iA-Loading-02GripperTakeDetection" )
      { S7_Templates := "SrcType := Int" } EQ_Contact(in1 := "AutoProcessData".A_ScanRotate.PartStatus, in2 := 0)
      { S7_Templates := "SrcType := Int" } EQ_Contact(in1 := "AutoProcessData".F_Robot1Grip1.PartStatus, in2 := 0)
      { S7_Templates := "SrcType := Int" } EQ_Contact(in1 := "AutoProcessData".F_Robot1Grip2.PartStatus, in2 := 0)
      { S7_Templates := "SrcType := Int" } EQ_Contact(in1 := "AutoProcessData".B_Press1.PartStatus, in2 := 0)
      Coil( "ChangeOver_DB".Robot_1.EmptyFinish )
   END_RUNG
   RUNG wire#w1
      { S7_Templates := "SrcType := Int" } EQ_Contact(in1 := "AutoProcessData".C_Glue.PartStatus, in2 := 0)
      { S7_Templates := "SrcType := Int" } EQ_Contact(in1 := "AutoProcessData".F_Robot2Grip1.PartStatus, in2 := 0)
      { S7_Templates := "SrcType := Int" } EQ_Contact(in1 := "AutoProcessData".F_Robot2Grip2.PartStatus, in2 := 0)
      { S7_Templates := "SrcType := Int" } EQ_Contact(in1 := "AutoProcessData".C_GlueNGBuffer.PartStatus, in2 := 0)
      { S7_Templates := "SrcType := Int" } EQ_Contact(in1 := "AutoProcessData".C_MagnScanNGBuffer.PartStatus, in2 := 0)
      { S7_Templates := "SrcType := Int" } EQ_Contact(in1 := "AutoProcessData".B_Press2.PartStatus, in2 := 0)
      I_Contact( "iA-Rotating product Check" )
      I_Contact( "iB-PressFitting-01ShaftDetection" )
      I_Contact( "iC-LocationShaftDetection" )
      I_Contact( "iB-PressFitting-02ShaftDetection" )
      Coil( "ChangeOver_DB".Robot_2.EmptyFinish )
   END_RUNG
   RUNG wire#w1
      { S7_Templates := "SrcType := Int" } EQ_Contact(in1 := "AutoProcessData".F_Robot3Grip1.PartStatus, in2 := 0)
      { S7_Templates := "SrcType := Int" } EQ_Contact(in1 := "AutoProcessData".F_Robot3Grip2.PartStatus, in2 := 0)
      Coil( "ChangeOver_DB".Robot_3.EmptyFinish )
   END_RUNG
   RUNG wire#w1
      Contact( "ChangeOver_DB".Robot_1.EmptyFinish )
      Contact( "ChangeOver_DB".Robot_2.EmptyFinish )
      Contact( "ChangeOver_DB".Robot_3.EmptyFinish )
      Coil( "ChangeOver_DB".Global.Station_empty )
   END_RUNG
   // the same network as SCL:
   "ChangeOver_DB".Robot_1.EmptyFinish := "AlwaysTRUE" AND NOT "iA-Loading-01GripperTakeDetection" AND NOT "iA-Loading-02GripperTakeDetection" AND ("AutoProcessData".A_ScanRotate.PartStatus = 0) AND ("AutoProcessData".F_Robot1Grip1.PartStatus = 0) AND ("AutoProcessData".F_Robot1Grip2.PartStatus = 0) AND ("AutoProcessData".B_Press1.PartStatus = 0);
   "ChangeOver_DB".Robot_2.EmptyFinish := "AlwaysTRUE" AND ("AutoProcessData".C_Glue.PartStatus = 0) AND ("AutoProcessData".F_Robot2Grip1.PartStatus = 0) AND ("AutoProcessData".F_Robot2Grip2.PartStatus = 0) AND ("AutoProcessData".C_GlueNGBuffer.PartStatus = 0) AND ("AutoProcessData".C_MagnScanNGBuffer.PartStatus = 0) AND ("AutoProcessData".B_Press2.PartStatus = 0) AND NOT "iA-Rotating product Check" AND NOT "iB-PressFitting-01ShaftDetection" AND NOT "iC-LocationShaftDetection" AND NOT "iB-PressFitting-02ShaftDetection";
   "ChangeOver_DB".Robot_3.EmptyFinish := "AlwaysTRUE" AND ("AutoProcessData".F_Robot3Grip1.PartStatus = 0) AND ("AutoProcessData".F_Robot3Grip2.PartStatus = 0);
   "ChangeOver_DB".Global.Station_empty := "AlwaysTRUE" AND "ChangeOver_DB".Robot_1.EmptyFinish AND "ChangeOver_DB".Robot_2.EmptyFinish AND "ChangeOver_DB".Robot_3.EmptyFinish;
END_REGION
END_FUNCTION
